// TwinCAT 3 PLC project TcUnit
// Title: TcUnit
// Company: www.tcunit.org
// Author: Jakob Sagatowski and contributors
// ProjectVersion: 1.0.1.1
// Description: TwinCAT unit testing framework. Documentation and examples are available at www.tcunit.org
// ProgramVersion: 3.1.4023.0
// libraries:
//   SysFile, * (System)
//   Tc2_Standard, * (Beckhoff Automation GmbH)
//   Tc2_System, * (Beckhoff Automation GmbH)
//   Tc2_Utilities, * (Beckhoff Automation GmbH)
//   Base Interfaces,newest,System
// project tree:
//   DUTs/ E_XmlError.TcDUT (not stored), ST_ADSLogStringMessage.TcDUT (not stored), ST_AssertResult.TcDUT (not stored), ST_AssertResultInstances.TcDUT (not stored), ST_AssertArrayResult.TcDUT (not stored), ST_AssertArrayResultInstances.TcDUT (not stored), U_ExpectedOrActual.TcDUT (not stored)
//   GVLs/ GVL_Param_TcUnit.TcGVL (not stored), GVL_Param_XmlControl.TcGVL (not stored), GVL_TcUnit.TcGVL (not stored)
//   ITFs/ I_AssertMessageFormatter.TcIO (not stored), I_TestResultFormatter.TcIO (not stored)
//   POUs/ FB_StringBuffer.TcPOU (not stored), FB_XmlControl.TcPOU (not stored), FB_FileControl.TcPOU (not stored), FB_AdjustAssertFailureMessageToMax252CharLength.TcPOU (not stored), FB_ADSAssertMessageFormatter.TcPOU (not stored), FB_ADSLogStringMessageFifoQueue.TcPOU (not stored), FB_ADSTestResultFormatter.TcPOU (not stored), FB_AnyComparator.TcPOU (not stored), FB_AssertResultStatic.TcPOU (not stored), FB_AssertArrayResultStatic.TcPOU (not stored), FB_TcUnitRunner.TcPOU (not stored), FB_Test.TcPOU (not stored), FB_TestSuite.TcPOU
//   POUs/Functions/ F_AnyToUnionValue.TcPOU (not stored), F_AnyTypeClassToString.TcPOU (not stored), F_IsAnyEqualToUnionValue.TcPOU (not stored), F_RemoveInstancePathAndProjectNameFromTestInstancePath.TcPOU (not stored), IS_TEST_FINISHED.TcPOU (not stored), RUN.TcPOU (not stored), TEST.TcPOU (not stored), TEST_FINISHED.TcPOU (not stored), TEST_FINISHED_NAMED.TcPOU (not stored)
//   POUs/Functions/WRITE_PROTECTED_/ WRITE_PROTECTED_BOOL.TcPOU (not stored), WRITE_PROTECTED_BYTE.TcPOU (not stored), WRITE_PROTECTED_DATE.TcPOU (not stored), WRITE_PROTECTED_DATE_AND_TIME.TcPOU (not stored), WRITE_PROTECTED_DINT.TcPOU (not stored), WRITE_PROTECTED_DWORD.TcPOU (not stored), WRITE_PROTECTED_INT.TcPOU (not stored), WRITE_PROTECTED_LREAL.TcPOU (not stored), WRITE_PROTECTED_REAL.TcPOU (not stored), WRITE_PROTECTED_SINT.TcPOU (not stored), WRITE_PROTECTED_STRING.TcPOU (not stored), WRITE_PROTECTED_TIME.TcPOU (not stored), WRITE_PROTECTED_TIME_OF_DAY.TcPOU (not stored), WRITE_PROTECTED_UDINT.TcPOU (not stored), WRITE_PROTECTED_UINT.TcPOU (not stored), WRITE_PROTECTED_USINT.TcPOU (not stored), WRITE_PROTECTED_WORD.TcPOU (not stored)
//   Version/ Global_Version.TcGVL

// ---- Version/Global_Version.TcGVL
{attribute 'TcGenerated'}
{attribute 'no-analysis'}
{attribute 'linkalways'}
// This function has been automatically generated from the project information.
VAR_GLOBAL CONSTANT
	{attribute 'const_non_replaced'}
	stLibVersion_TcUnit : ST_LibVersion := (iMajor := 1, iMinor := 0, iBuild := 1, iRevision := 1, nFlags := 0, sVersion := '1.0.1.1');
END_VAR

// ---- POUs/FB_TestSuite.TcPOU
(* This function block is responsible for holding the internal state of the test suite.
   Every test suite can have one or more tests, and every test can do one or more asserts.
   It's also responsible for providing all the assert-methods for asserting different data types.
   Only failed assertions are recorded.
*)
{attribute 'call_after_init'}
{attribute 'reflection'}
FUNCTION_BLOCK FB_TestSuite
VAR
    {attribute 'instance-path'}
    {attribute 'noinit'}
    InstancePath : Tc2_System.T_MaxString;

    (* We need to have access to specific information of the current task that this test suite
       is executed in. This is for instance necessary when we need to know whether a test is
       defined already. The definition of a test that is defined already is that we call on it
       with the same name twice in the same cycle *)
    GetCurrentTaskIndex : Tc2_System.GETCURTASKINDEX;

    NumberOfTests : UINT := 0;
    Tests : ARRAY[1..GVL_Param_TcUnit.MaxNumberOfTestsForEachTestSuite] OF FB_Test;
    (* Rising trigger of whether we have already notified the user of that the test name pointed to by the current
       position is a duplicate *)
    TestDuplicateNameTrigger : ARRAY[1..GVL_Param_TcUnit.MaxNumberOfTestsForEachTestSuite] OF Tc2_Standard.R_TRIG;
    (* Last cycle count index for a specific test. Used to detect whether this test has already been defined in the
       current test suite *)
    TestCycleCountIndex : ARRAY[1..GVL_Param_TcUnit.MaxNumberOfTestsForEachTestSuite] OF UDINT;

    AssertResults : FB_AssertResultStatic;
    AssertArrayResult : FB_AssertArrayResultStatic;

    (* Prints the failed asserts to ADS so that Visual Studio can display the assert message.
       This assert formatter can be replaced with something else than ADS *)
    ADSAssertMessageFormatter : FB_ADSAssertMessageFormatter;
    AssertMessageFormatter : I_AssertMessageFormatter := ADSAssertMessageFormatter;
END_VAR

METHOD PUBLIC AddTest
VAR_INPUT
    TestName : Tc2_System.T_MaxString;
END_VAR
VAR
    IteratorCounter : UINT;
    ErrorMessage : Tc2_System.T_MaxString;
    TestInstancePath : Tc2_System.T_MaxString;
    FunctionCallResult : DINT;
    CycleCount : UDINT;
    TestWithThisNameAlreadyExists : BOOL := FALSE;
    LowerCasedTestName : Tc2_System.T_MaxString;
    TrimmedTestName : Tc2_System.T_MaxString;
END_VAR
GVL_TcUnit.IgnoreCurrentTest := FALSE; // Reset the ignore current test flag

TrimmedTestName := Tc2_Utilities.F_LTrim(in := TestName);
TrimmedTestName := Tc2_Utilities.F_RTrim(in := TrimmedTestName);
LowerCasedTestName := Tc2_Utilities.F_ToLCase(in := TrimmedTestName);

(* Check if this test should be disabled *)
IF Tc2_Utilities.FIND(STR1 := LowerCasedTestName, STR2 := 'disabled_') = 1 THEN
    GVL_TcUnit.IgnoreCurrentTest := TRUE;
    RETURN;
END_IF

GetCurrentTaskIndex(); // Gets the task index of where this function block instance is being run in

(* Check if the test name already exists. Make sure there are no other tests with the same name already
   added for this test suite *)

CycleCount := TwinCAT_SystemInfoVarList._TaskInfo[GetCurrentTaskIndex.index].CycleCount;

(* Iterate all the test names that up to this point have been added for this test suite *)
FOR IteratorCounter := 1 TO NumberOfTests BY 1 DO
    IF Tests[IteratorCounter].GetName() = TrimmedTestName THEN
        TestWithThisNameAlreadyExists := TRUE;
        (* Check if a test with this name has already been called in this PLC cycle *)
        IF TestCycleCountIndex[IteratorCounter] = CycleCount THEN
            GVL_TcUnit.IgnoreCurrentTest := TRUE;
            (* A test with this name already exists for this test suite and has already been called in this cycle.
               Send a message notification, but only if we have not done so already. *)
            TestDuplicateNameTrigger[IteratorCounter](CLK := TRUE);
            IF TestDuplicateNameTrigger[IteratorCounter].Q THEN // Rising edge detected. We have not reported this before
                TestInstancePath := F_RemoveInstancePathAndProjectNameFromTestInstancePath(TestInstancePath :=
                                                                                           GVL_TcUnit.CurrentTestSuiteBeingCalled^.GetInstancePath());
                ErrorMessage := 'Test with name $'%s$' already exists in test suite $'';
                ErrorMessage := Tc2_Standard.CONCAT(STR1 := ErrorMessage, STR2 := TestInstancePath);
                ErrorMessage := Tc2_Standard.CONCAT(STR1 := ErrorMessage, STR2 := '$'');
                GVL_TcUnit.AdsLogger.WriteLog(MsgFmtStr := ErrorMessage,
                                              StrArg := TrimmedTestName);
            END_IF
        END_IF
        TestCycleCountIndex[IteratorCounter] := CycleCount;
    END_IF
END_FOR

IF NOT TestWithThisNameAlreadyExists THEN
    (* Test has not been found. Add it. *)
    Tests[IteratorCounter].SetName(Name := TrimmedTestName);
    NumberOfTests := NumberOfTests + 1;
    TestCycleCountIndex[NumberOfTests] := CycleCount;
END_IF
END_METHOD

METHOD PRIVATE AddTestNameToInstancePath : Tc2_System.T_MaxString
VAR_INPUT
    TestInstancePath : Tc2_System.T_MaxString;
END_VAR
VAR
    CompleteTestInstancePath : Tc2_System.T_MaxString;
END_VAR
CompleteTestInstancePath := Tc2_Utilities.CONCAT(STR1 := TestInstancePath, STR2 := '@');
AddTestNameToInstancePath := Tc2_Utilities.CONCAT(STR1 := CompleteTestInstancePath, STR2 := GVL_TcUnit.CurrentTestNameBeingCalled);
END_METHOD

METHOD PUBLIC AreAllTestsFinished : BOOL
VAR
    Counter : UINT;

    GetCurTaskIndex : Tc2_System.GETCURTASKINDEX;
END_VAR
AreAllTestsFinished := FALSE;

IF NumberOfTests > 0 THEN
    AreAllTestsFinished := TRUE;
    FOR Counter := 1 TO GetNumberOfTests() BY 1 DO
        AreAllTestsFinished := AreAllTestsFinished AND Tests[Counter].IsFinished();
    END_FOR
END_IF

(* If we have been running at least one cycle and no tests are registered it means that this testsuite is empty
   and doesn't contain any test cases. In that case, add a warning message and ignore this testsuite. *)
GetCurTaskIndex();
IF NumberOfTests = 0 AND NOT TwinCAT_SystemInfoVarList._TaskInfo[GetCurTaskIndex.index].FirstCycle THEN
    AreAllTestsFinished := TRUE;
END_IF
END_METHOD

METHOD PUBLIC AssertArray2dEquals_LREAL
VAR_IN_OUT
    Expecteds : ARRAY[*,*] OF LREAL; // LREAL 2d array with expected values
    Actuals : ARRAY[*,*] OF LREAL; // LREAL 2d array with actual values
END_VAR
VAR_INPUT
    Delta : LREAL; // The maximum delta between the value of expected and actual for which both numbers are still considered equal, proportional to the Expected value in that array cell
    Message : Tc2_System.T_MaxString; // The identifying message for the assertion error
END_VAR
VAR
    Equals : BOOL := TRUE;
    SizeEquals : BOOL := TRUE;
    ExpectedString : STRING;
    ActualString : STRING;
    AlreadyReported : BOOL;
    TestInstancePath : Tc2_System.T_MaxString;
    DimensionIndex : USINT; // Index when looping through Dimensions
    LowerBoundExpecteds : ARRAY[1..2] OF DINT; // Lower bounds of Expecteds array in each dimension
    UpperBoundExpecteds : ARRAY[1..2] OF DINT; // Upper bounds of Expecteds array in each dimension
    LowerBoundActuals : ARRAY[1..2] OF DINT; // Lower bounds of Actuals array in each dimension
    UpperBoundActuals : ARRAY[1..2] OF DINT; // Upper bounds of Actuals array in each dimension
    SizeOfExpecteds : ARRAY[1..2] OF DINT; // Size of Expecteds array in each dimension
    SizeOfActuals : ARRAY[1..2] OF DINT; // Size of Actuals array in each dimension
    Offset : ARRAY[1..2] OF DINT; // Current Array index offsets from Lower Bound in each dimension
    ExpectedArrayIndex : ARRAY[1..2] OF DINT; // Array of current Expected array indexes when looping through arrays
    ActualArrayIndex : ARRAY[1..2] OF DINT; // Array of current Actual array indexes when looping through arrays
    Expected : LREAL; // Single expected value
    Actual : LREAL; // Single actual value
END_VAR
IF GVL_TcUnit.IgnoreCurrentTest OR GVL_TcUnit.CurrentTestIsFinished THEN
    RETURN;
END_IF

TestInstancePath := AddTestNameToInstancePath(FindTestSuiteInstancePath());

(* UPPER_BOUND and LOWER_BOUND require literals for their second parameter,
   so they can't be called in a dimension-based loop.
   Thus we copy the array dimensions into arrays which accept variable indexes *)
LowerBoundExpecteds[1] := LOWER_BOUND(Expecteds, 1);
UpperBoundExpecteds[1] := UPPER_BOUND(Expecteds, 1);
LowerBoundExpecteds[2] := LOWER_BOUND(Expecteds, 2);
UpperBoundExpecteds[2] := UPPER_BOUND(Expecteds, 2);
LowerBoundActuals[1] := LOWER_BOUND(Actuals, 1);
UpperBoundActuals[1] := UPPER_BOUND(Actuals, 1);
LowerBoundActuals[2] := LOWER_BOUND(Actuals, 2);
UpperBoundActuals[2] := UPPER_BOUND(Actuals, 2);

FOR DimensionIndex := 1 TO 2 DO
    SizeOfExpecteds[DimensionIndex] := ABS(UpperBoundExpecteds[DimensionIndex] - LowerBoundExpecteds[DimensionIndex]) + 1;
    SizeOfActuals[DimensionIndex] := ABS(UpperBoundActuals[DimensionIndex] - LowerBoundActuals[DimensionIndex]) + 1;

    IF SizeOfExpecteds[DimensionIndex] <> SizeOfActuals[DimensionIndex] THEN
        Equals := FALSE;
        SizeEquals := FALSE;
    END_IF
END_FOR

IF SizeEquals THEN
    (* Even though we know that both arrays are equal in size, the two arrays can start at two completely different
       indexes in each dimension, which needs to be taken into account. *)
    FOR Offset[1] := 0 TO SizeOfExpecteds[1] - 1 DO // Iterate Dimension 1
        FOR Offset[2] := 0 TO SizeOfExpecteds[2] - 1 DO // Iterate Dimension 2
            // Update index variables
            FOR DimensionIndex := 1 TO 2 DO
                ExpectedArrayIndex[DimensionIndex] := LowerBoundExpecteds[DimensionIndex] + Offset[DimensionIndex];
                ActualArrayIndex[DimensionIndex] := LowerBoundActuals[DimensionIndex] + Offset[DimensionIndex];
            END_FOR

            // Get array element values
            Expected := Expecteds[ExpectedArrayIndex[1], ExpectedArrayIndex[2]];
            Actual := Actuals[ActualArrayIndex[1], ActualArrayIndex[2]]; 

            IF ABS(Expected - Actual) > Delta THEN
                Equals := FALSE;
                EXIT;
            END_IF
        END_FOR

        // Check for loop bailout
        IF NOT Equals THEN
            EXIT;
        END_IF
    END_FOR
END_IF

IF NOT Equals THEN
    AssertArrayResult.ReportResult(ExpectedsSize := DINT_TO_UDINT(SizeOfExpecteds[1] * SizeOfExpecteds[2]),
                                   ExpectedsTypeClass := IBaseLibrary.TypeClass.TYPE_LREAL,
                                   ActualsSize := DINT_TO_UDINT(SizeOfActuals[1] * SizeOfActuals[2]),
                                   ActualsTypeClass := IBaseLibrary.TypeClass.TYPE_LREAL,
                                   Message := Message,
                                   TestInstancePath := TestInstancePath,
                                   AlreadyReported => AlreadyReported);
END_IF

IF NOT AlreadyReported AND NOT Equals THEN
    SetTestFailed();

    IF NOT SizeEquals THEN
        Message := Tc2_Standard.CONCAT(STR1 := Message, STR2 := ', size of arrays not matching.');
        ExpectedString := 'SIZE = [';
        ExpectedString := Tc2_Standard.CONCAT(STR1 := ExpectedString, STR2 := DINT_TO_STRING(LowerBoundExpecteds[1]));
        ExpectedString := Tc2_Standard.CONCAT(STR1 := ExpectedString, STR2 := '..');
        ExpectedString := Tc2_Standard.CONCAT(STR1 := ExpectedString, STR2 := DINT_TO_STRING(UpperBoundExpecteds[1]));
        ExpectedString := Tc2_Standard.CONCAT(STR1 := ExpectedString, STR2 := ',');
        ExpectedString := Tc2_Standard.CONCAT(STR1 := ExpectedString, STR2 := DINT_TO_STRING(LowerBoundExpecteds[2]));
        ExpectedString := Tc2_Standard.CONCAT(STR1 := ExpectedString, STR2 := '..');
        ExpectedString := Tc2_Standard.CONCAT(STR1 := ExpectedString, STR2 := DINT_TO_STRING(UpperBoundExpecteds[2]));
        ExpectedString := Tc2_Standard.CONCAT(STR1 := ExpectedString, STR2 := '] (');
        ExpectedString := Tc2_Standard.CONCAT(STR1 := ExpectedString, STR2 := DINT_TO_STRING(SizeOfExpecteds[1]));
        ExpectedString := Tc2_Standard.CONCAT(STR1 := ExpectedString, STR2 := 'x');
        ExpectedString := Tc2_Standard.CONCAT(STR1 := ExpectedString, STR2 := DINT_TO_STRING(SizeOfExpecteds[2]));
        ExpectedString := Tc2_Standard.CONCAT(STR1 := ExpectedString, STR2 := ')');

        ActualString := 'SIZE = [';
        ActualString := Tc2_Standard.CONCAT(STR1 := ActualString, STR2 := DINT_TO_STRING(LowerBoundActuals[1]));
        ActualString := Tc2_Standard.CONCAT(STR1 := ActualString, STR2 := '..');
        ActualString := Tc2_Standard.CONCAT(STR1 := ActualString, STR2 := DINT_TO_STRING(UpperBoundActuals[1]));
        ActualString := Tc2_Standard.CONCAT(STR1 := ActualString, STR2 := ',');
        ActualString := Tc2_Standard.CONCAT(STR1 := ActualString, STR2 := DINT_TO_STRING(LowerBoundActuals[2]));
        ActualString := Tc2_Standard.CONCAT(STR1 := ActualString, STR2 := '..');
        ActualString := Tc2_Standard.CONCAT(STR1 := ActualString, STR2 := DINT_TO_STRING(UpperBoundActuals[2]));
        ActualString := Tc2_Standard.CONCAT(STR1 := ActualString, STR2 := '] (');
        ActualString := Tc2_Standard.CONCAT(STR1 := ActualString, STR2 := DINT_TO_STRING(SizeOfActuals[1]));
        ActualString := Tc2_Standard.CONCAT(STR1 := ActualString, STR2 := 'x');
        ActualString := Tc2_Standard.CONCAT(STR1 := ActualString, STR2 := DINT_TO_STRING(SizeOfActuals[2]));
        ActualString := Tc2_Standard.CONCAT(STR1 := ActualString, STR2 := ')');
    ELSE
        ExpectedString := 'ARRAY[';
        ExpectedString := Tc2_Standard.CONCAT(STR1 := ExpectedString, STR2 := DINT_TO_STRING(ExpectedArrayIndex[1]));
        ExpectedString := Tc2_Standard.CONCAT(STR1 := ExpectedString, STR2 := ',');
        ExpectedString := Tc2_Standard.CONCAT(STR1 := ExpectedString, STR2 := DINT_TO_STRING(ExpectedArrayIndex[2]));
        ExpectedString := Tc2_Standard.CONCAT(STR1 := ExpectedString, STR2 := '] = ');
        ExpectedString := Tc2_Standard.CONCAT(STR1 := ExpectedString, STR2 := LREAL_TO_STRING(Expected));

        ActualString := 'ARRAY[';
        ActualString := Tc2_Standard.CONCAT(STR1 := ActualString, STR2 := DINT_TO_STRING(ActualArrayIndex[1]));
        ActualString := Tc2_Standard.CONCAT(STR1 := ActualString, STR2 := ',');
        ActualString := Tc2_Standard.CONCAT(STR1 := ActualString, STR2 := DINT_TO_STRING(ActualArrayIndex[2]));
        ActualString := Tc2_Standard.CONCAT(STR1 := ActualString, STR2 := '] = ');
        ActualString := Tc2_Standard.CONCAT(STR1 := ActualString, STR2 := LREAL_TO_STRING(Actual));
    END_IF

    AssertMessageFormatter.LogAssertFailure(Expected := ExpectedString,
                                            Actual := ActualString,
                                            Message := Message,
                                            TestInstancePath := TestInstancePath);
END_IF
END_METHOD

METHOD PUBLIC AssertArray2dEquals_REAL
VAR_IN_OUT
    Expecteds : ARRAY[*,*] OF REAL; // REAL 2d array with expected values
    Actuals : ARRAY[*,*] OF REAL; // REAL 2d array with actual values
END_VAR
VAR_INPUT
    Delta : REAL; // The maximum delta between the value of expected and actual for which both numbers are still considered equal, proportional to the Expected value in that array cell
    Message : Tc2_System.T_MaxString; // The identifying message for the assertion error
END_VAR
VAR
    Equals : BOOL := TRUE;
    SizeEquals : BOOL := TRUE;
    ExpectedString : STRING;
    ActualString : STRING;
    AlreadyReported : BOOL;
    TestInstancePath : Tc2_System.T_MaxString;
    DimensionIndex : USINT; // Index when looping through Dimensions
    LowerBoundExpecteds : ARRAY[1..2] OF DINT; // Lower bounds of Expecteds array in each dimension
    UpperBoundExpecteds : ARRAY[1..2] OF DINT; // Upper bounds of Expecteds array in each dimension
    LowerBoundActuals : ARRAY[1..2] OF DINT; // Lower bounds of Actuals array in each dimension
    UpperBoundActuals : ARRAY[1..2] OF DINT; // Upper bounds of Actuals array in each dimension
    SizeOfExpecteds : ARRAY[1..2] OF DINT; // Size of Expecteds array in each dimension
    SizeOfActuals : ARRAY[1..2] OF DINT; // Size of Actuals array in each dimension
    Offset : ARRAY[1..2] OF DINT; // Current Array index offsets from Lower Bound in each dimension
    ExpectedArrayIndex : ARRAY[1..2] OF DINT; // Array of current Expected array indexes when looping through arrays
    ActualArrayIndex : ARRAY[1..2] OF DINT; // Array of current Actual array indexes when looping through arrays
    Expected : REAL; // Single expected value
    Actual : REAL; // Single actual value
END_VAR
IF GVL_TcUnit.IgnoreCurrentTest OR GVL_TcUnit.CurrentTestIsFinished THEN
    RETURN;
END_IF

TestInstancePath := AddTestNameToInstancePath(FindTestSuiteInstancePath());

(* UPPER_BOUND and LOWER_BOUND require literals for their second parameter, 
   so they can't be called in a dimension-based loop.
   Thus we copy the ARRAY dimensions into arrays which accept variable indexes *)
LowerBoundExpecteds[1] := LOWER_BOUND(Expecteds, 1);
UpperBoundExpecteds[1] := UPPER_BOUND(Expecteds, 1);
LowerBoundExpecteds[2] := LOWER_BOUND(Expecteds, 2);
UpperBoundExpecteds[2] := UPPER_BOUND(Expecteds, 2);
LowerBoundActuals[1] := LOWER_BOUND(Actuals, 1);
UpperBoundActuals[1] := UPPER_BOUND(Actuals, 1);
LowerBoundActuals[2] := LOWER_BOUND(Actuals, 2);
UpperBoundActuals[2] := UPPER_BOUND(Actuals, 2);

FOR DimensionIndex := 1 TO 2 DO
    SizeOfExpecteds[DimensionIndex] := ABS(UpperBoundExpecteds[DimensionIndex] - LowerBoundExpecteds[DimensionIndex]) + 1;
    SizeOfActuals[DimensionIndex] := ABS(UpperBoundActuals[DimensionIndex] - LowerBoundActuals[DimensionIndex]) + 1;

    IF SizeOfExpecteds[DimensionIndex] <> SizeOfActuals[DimensionIndex] THEN
        Equals := FALSE;
        SizeEquals := FALSE;
    END_IF
END_FOR

IF SizeEquals THEN
    (* Even though we know that both arrays are equal in size, the two arrays can start at two completely different
       indexes in each dimension, which needs to be taken into account. *)
    FOR Offset[1] := 0 TO SizeOfExpecteds[1] - 1 DO // Iterate Dimension 1
        FOR Offset[2] := 0 TO SizeOfExpecteds[2] - 1 DO // Iterate Dimension 2
            // Update index variables
            FOR DimensionIndex := 1 TO 2 DO
                ExpectedArrayIndex[DimensionIndex] := LowerBoundExpecteds[DimensionIndex] + Offset[DimensionIndex];
                ActualArrayIndex[DimensionIndex] := LowerBoundActuals[DimensionIndex] + Offset[DimensionIndex];
            END_FOR

            // Get array element values
            Expected := Expecteds[ExpectedArrayIndex[1], ExpectedArrayIndex[2]];
            Actual := Actuals[ActualArrayIndex[1], ActualArrayIndex[2]]; 

            IF ABS(Expected - Actual) > Delta THEN
                Equals := FALSE;
                EXIT;
            END_IF
        END_FOR

        // Check for loop bailout
        IF NOT Equals THEN
            EXIT;
        END_IF
    END_FOR
END_IF

IF NOT Equals THEN
    AssertArrayResult.ReportResult(ExpectedsSize := DINT_TO_UDINT(SizeOfExpecteds[1] * SizeOfExpecteds[2]),
                                   ExpectedsTypeClass := IBaseLibrary.TypeClass.TYPE_REAL,
                                   ActualsSize := DINT_TO_UDINT(SizeOfActuals[1] * SizeOfActuals[2]),
                                   ActualsTypeClass := IBaseLibrary.TypeClass.TYPE_REAL,
                                   Message := Message,
                                   TestInstancePath := TestInstancePath,
                                   AlreadyReported => AlreadyReported);
END_IF

IF NOT AlreadyReported AND NOT Equals THEN
    SetTestFailed();

    IF NOT SizeEquals THEN
        Message := Tc2_Standard.CONCAT(STR1 := Message, STR2 := ', size of arrays not matching.');
        ExpectedString := 'SIZE = [';
        ExpectedString := Tc2_Standard.CONCAT(STR1 := ExpectedString, STR2 := DINT_TO_STRING(LowerBoundExpecteds[1]));
        ExpectedString := Tc2_Standard.CONCAT(STR1 := ExpectedString, STR2 := '..');
        ExpectedString := Tc2_Standard.CONCAT(STR1 := ExpectedString, STR2 := DINT_TO_STRING(UpperBoundExpecteds[1]));
        ExpectedString := Tc2_Standard.CONCAT(STR1 := ExpectedString, STR2 := ',');
        ExpectedString := Tc2_Standard.CONCAT(STR1 := ExpectedString, STR2 := DINT_TO_STRING(LowerBoundExpecteds[2]));
        ExpectedString := Tc2_Standard.CONCAT(STR1 := ExpectedString, STR2 := '..');
        ExpectedString := Tc2_Standard.CONCAT(STR1 := ExpectedString, STR2 := DINT_TO_STRING(UpperBoundExpecteds[2]));
        ExpectedString := Tc2_Standard.CONCAT(STR1 := ExpectedString, STR2 := '] (');
        ExpectedString := Tc2_Standard.CONCAT(STR1 := ExpectedString, STR2 := DINT_TO_STRING(SizeOfExpecteds[1]));
        ExpectedString := Tc2_Standard.CONCAT(STR1 := ExpectedString, STR2 := 'x');
        ExpectedString := Tc2_Standard.CONCAT(STR1 := ExpectedString, STR2 := DINT_TO_STRING(SizeOfExpecteds[2]));
        ExpectedString := Tc2_Standard.CONCAT(STR1 := ExpectedString, STR2 := ')');

        ActualString := 'SIZE = [';
        ActualString := Tc2_Standard.CONCAT(STR1 := ActualString, STR2 := DINT_TO_STRING(LowerBoundActuals[1]));
        ActualString := Tc2_Standard.CONCAT(STR1 := ActualString, STR2 := '..');
        ActualString := Tc2_Standard.CONCAT(STR1 := ActualString, STR2 := DINT_TO_STRING(UpperBoundActuals[1]));
        ActualString := Tc2_Standard.CONCAT(STR1 := ActualString, STR2 := ',');
        ActualString := Tc2_Standard.CONCAT(STR1 := ActualString, STR2 := DINT_TO_STRING(LowerBoundActuals[2]));
        ActualString := Tc2_Standard.CONCAT(STR1 := ActualString, STR2 := '..');
        ActualString := Tc2_Standard.CONCAT(STR1 := ActualString, STR2 := DINT_TO_STRING(UpperBoundActuals[2]));
        ActualString := Tc2_Standard.CONCAT(STR1 := ActualString, STR2 := '] (');
        ActualString := Tc2_Standard.CONCAT(STR1 := ActualString, STR2 := DINT_TO_STRING(SizeOfActuals[1]));
        ActualString := Tc2_Standard.CONCAT(STR1 := ActualString, STR2 := 'x');
        ActualString := Tc2_Standard.CONCAT(STR1 := ActualString, STR2 := DINT_TO_STRING(SizeOfActuals[2]));
        ActualString := Tc2_Standard.CONCAT(STR1 := ActualString, STR2 := ')');
    ELSE
        ExpectedString := 'ARRAY[';
        ExpectedString := Tc2_Standard.CONCAT(STR1 := ExpectedString, STR2 := DINT_TO_STRING(ExpectedArrayIndex[1]));
        ExpectedString := Tc2_Standard.CONCAT(STR1 := ExpectedString, STR2 := ',');
        ExpectedString := Tc2_Standard.CONCAT(STR1 := ExpectedString, STR2 := DINT_TO_STRING(ExpectedArrayIndex[2]));
        ExpectedString := Tc2_Standard.CONCAT(STR1 := ExpectedString, STR2 := '] = ');
        ExpectedString := Tc2_Standard.CONCAT(STR1 := ExpectedString, STR2 := REAL_TO_STRING(Expected));

        ActualString := 'ARRAY[';
        ActualString := Tc2_Standard.CONCAT(STR1 := ActualString, STR2 := DINT_TO_STRING(ActualArrayIndex[1]));
        ActualString := Tc2_Standard.CONCAT(STR1 := ActualString, STR2 := ',');
        ActualString := Tc2_Standard.CONCAT(STR1 := ActualString, STR2 := DINT_TO_STRING(ActualArrayIndex[2]));
        ActualString := Tc2_Standard.CONCAT(STR1 := ActualString, STR2 := '] = ');
        ActualString := Tc2_Standard.CONCAT(STR1 := ActualString, STR2 := REAL_TO_STRING(Actual));
    END_IF

    AssertMessageFormatter.LogAssertFailure(Expected := ExpectedString,
                                            Actual := ActualString,
                                            Message := Message,
                                            TestInstancePath := TestInstancePath);
END_IF
END_METHOD

METHOD PUBLIC AssertArray3dEquals_LREAL
VAR_IN_OUT
    Expecteds : ARRAY[*,*,*] OF LREAL; // LREAL 3d array with expected values
    Actuals : ARRAY[*,*,*] OF LREAL; // LREAL 3d array with actual values
END_VAR
VAR_INPUT
    Delta : LREAL;  // The maximum delta between the value of expected and actual for which both numbers are still considered equal, proportional to the Expected value in that array cell
    Message : Tc2_System.T_MaxString; // The identifying message for the assertion error
END_VAR
VAR
    Equals : BOOL := TRUE;
    SizeEquals : BOOL := TRUE;
    ExpectedString : STRING;
    ActualString : STRING;
    AlreadyReported : BOOL;
    TestInstancePath : Tc2_System.T_MaxString;
    DimensionIndex : USINT;  // Index when looping through Dimensions
    LowerBoundExpecteds : ARRAY[1..3] OF DINT; // Lower bounds of Expecteds array in each dimension
    UpperBoundExpecteds : ARRAY[1..3] OF DINT; // Upper bounds of Expecteds array in each dimension
    LowerBoundActuals : ARRAY[1..3] OF DINT; // Lower bounds of Actuals array in each dimension
    UpperBoundActuals : ARRAY[1..3] OF DINT; // Upper bounds of Actuals array in each dimension
    SizeOfExpecteds : ARRAY[1..3] OF DINT; // Size of Expecteds array in each dimension
    SizeOfActuals : ARRAY[1..3] OF DINT; // Size of Actuals array in each dimension
    Offset : ARRAY[1..3] OF DINT; // Current Array index offsets from Lower Bound in each dimension
    ExpectedArrayIndex : ARRAY[1..3] OF DINT; // Array of current Expected array indexes when looping through arrays
    ActualArrayIndex : ARRAY[1..3] OF DINT; // Array of current Actual array indexes when looping through arrays
    Expected : LREAL; // Single expected value
    Actual : LREAL; // Single actual value
END_VAR
IF GVL_TcUnit.IgnoreCurrentTest OR GVL_TcUnit.CurrentTestIsFinished THEN
    RETURN;
END_IF

TestInstancePath := AddTestNameToInstancePath(FindTestSuiteInstancePath());

(* UPPER_BOUND and LOWER_BOUND require literals for their second parameter,
   so they can't be called in a dimension-based loop.
   Thus we copy the array dimensions into arrays which accept variable indexes *)
LowerBoundExpecteds[1] := LOWER_BOUND(Expecteds, 1);
UpperBoundExpecteds[1] := UPPER_BOUND(Expecteds, 1);
LowerBoundExpecteds[2] := LOWER_BOUND(Expecteds, 2);
UpperBoundExpecteds[2] := UPPER_BOUND(Expecteds, 2);
LowerBoundExpecteds[3] := LOWER_BOUND(Expecteds, 3);
UpperBoundExpecteds[3] := UPPER_BOUND(Expecteds, 3);
LowerBoundActuals[1] := LOWER_BOUND(Actuals, 1);
UpperBoundActuals[1] := UPPER_BOUND(Actuals, 1);
LowerBoundActuals[2] := LOWER_BOUND(Actuals, 2);
UpperBoundActuals[2] := UPPER_BOUND(Actuals, 2);
LowerBoundActuals[3] := LOWER_BOUND(Actuals, 3);
UpperBoundActuals[3] := UPPER_BOUND(Actuals, 3);

FOR DimensionIndex := 1 TO 3 DO
    SizeOfExpecteds[DimensionIndex] := ABS(UpperBoundExpecteds[DimensionIndex] - LowerBoundExpecteds[DimensionIndex]) + 1;
    SizeOfActuals[DimensionIndex] := ABS(UpperBoundActuals[DimensionIndex] - LowerBoundActuals[DimensionIndex]) + 1;

    IF SizeOfExpecteds[DimensionIndex] <> SizeOfActuals[DimensionIndex] THEN
        Equals := FALSE;
        SizeEquals := FALSE;
    END_IF
END_FOR

IF SizeEquals THEN
    (* Even though we know that both arrays are equal in size, the three arrays can start at three completely different
       indexes in each dimension, which needs to be taken into account. *)
    FOR Offset[1] := 0 TO SizeOfExpecteds[1] - 1 DO // Iterate Dimension 1
        FOR Offset[2] := 0 TO SizeOfExpecteds[2] - 1 DO // Iterate Dimension 2
            FOR Offset[3] := 0 TO SizeOfExpecteds[3] - 1 DO // Iterate Dimension 3
                // Update index variables
                FOR DimensionIndex := 1 TO 3 DO
                    ExpectedArrayIndex[DimensionIndex] := LowerBoundExpecteds[DimensionIndex] + Offset[DimensionIndex];
                    ActualArrayIndex[DimensionIndex] := LowerBoundActuals[DimensionIndex] + Offset[DimensionIndex];
                END_FOR

                // Get array element values
                Expected := Expecteds[ExpectedArrayIndex[1], ExpectedArrayIndex[2], ExpectedArrayIndex[3]];
                Actual := Actuals[ActualArrayIndex[1], ActualArrayIndex[2], ActualArrayIndex[3]]; 

                IF ABS(Expected - Actual) > Delta THEN
                    Equals := FALSE;
                    EXIT;
                END_IF
            END_FOR

            // Check for loop bailout
            IF NOT Equals THEN
                EXIT;
            END_IF
        END_FOR

        // Check for loop bailout
        IF NOT Equals THEN
            EXIT;
        END_IF
    END_FOR
END_IF

IF NOT Equals THEN
    AssertArrayResult.ReportResult(ExpectedsSize := DINT_TO_UDINT(SizeOfExpecteds[1] * SizeOfExpecteds[2] * SizeOfExpecteds[3]),
                                   ExpectedsTypeClass := IBaseLibrary.TypeClass.TYPE_LREAL,
                                   ActualsSize := DINT_TO_UDINT(SizeOfActuals[1] * SizeOfActuals[2] * SizeOfActuals[3]),
                                   ActualsTypeClass := IBaseLibrary.TypeClass.TYPE_LREAL,
                                   Message := Message,
                                   TestInstancePath := TestInstancePath,
                                   AlreadyReported => AlreadyReported);
END_IF

IF NOT AlreadyReported AND NOT Equals THEN
    SetTestFailed();

    IF NOT SizeEquals THEN
        Message := Tc2_Standard.CONCAT(STR1 := Message, STR2 := ', size of arrays not matching.');
        ExpectedString := 'SIZE = [';
        ExpectedString := Tc2_Standard.CONCAT(STR1 := ExpectedString, STR2 := DINT_TO_STRING(LowerBoundExpecteds[1]));
        ExpectedString := Tc2_Standard.CONCAT(STR1 := ExpectedString, STR2 := '..');
        ExpectedString := Tc2_Standard.CONCAT(STR1 := ExpectedString, STR2 := DINT_TO_STRING(UpperBoundExpecteds[1]));
        ExpectedString := Tc2_Standard.CONCAT(STR1 := ExpectedString, STR2 := ',');
        ExpectedString := Tc2_Standard.CONCAT(STR1 := ExpectedString, STR2 := DINT_TO_STRING(LowerBoundExpecteds[2]));
        ExpectedString := Tc2_Standard.CONCAT(STR1 := ExpectedString, STR2 := '..');
        ExpectedString := Tc2_Standard.CONCAT(STR1 := ExpectedString, STR2 := DINT_TO_STRING(UpperBoundExpecteds[2]));
        ExpectedString := Tc2_Standard.CONCAT(STR1 := ExpectedString, STR2 := ',');
        ExpectedString := Tc2_Standard.CONCAT(STR1 := ExpectedString, STR2 := DINT_TO_STRING(LowerBoundExpecteds[3]));
        ExpectedString := Tc2_Standard.CONCAT(STR1 := ExpectedString, STR2 := '..');
        ExpectedString := Tc2_Standard.CONCAT(STR1 := ExpectedString, STR2 := DINT_TO_STRING(UpperBoundExpecteds[3]));
        ExpectedString := Tc2_Standard.CONCAT(STR1 := ExpectedString, STR2 := '] (');
        ExpectedString := Tc2_Standard.CONCAT(STR1 := ExpectedString, STR2 := DINT_TO_STRING(SizeOfExpecteds[1]));
        ExpectedString := Tc2_Standard.CONCAT(STR1 := ExpectedString, STR2 := 'x');
        ExpectedString := Tc2_Standard.CONCAT(STR1 := ExpectedString, STR2 := DINT_TO_STRING(SizeOfExpecteds[2]));
        ExpectedString := Tc2_Standard.CONCAT(STR1 := ExpectedString, STR2 := 'x');
        ExpectedString := Tc2_Standard.CONCAT(STR1 := ExpectedString, STR2 := DINT_TO_STRING(SizeOfExpecteds[3]));
        ExpectedString := Tc2_Standard.CONCAT(STR1 := ExpectedString, STR2 := ')');

        ActualString := 'SIZE = [';
        ActualString := Tc2_Standard.CONCAT(STR1 := ActualString, STR2 := DINT_TO_STRING(LowerBoundActuals[1]));
        ActualString := Tc2_Standard.CONCAT(STR1 := ActualString, STR2 := '..');
        ActualString := Tc2_Standard.CONCAT(STR1 := ActualString, STR2 := DINT_TO_STRING(UpperBoundActuals[1]));
        ActualString := Tc2_Standard.CONCAT(STR1 := ActualString, STR2 := ',');
        ActualString := Tc2_Standard.CONCAT(STR1 := ActualString, STR2 := DINT_TO_STRING(LowerBoundActuals[2]));
        ActualString := Tc2_Standard.CONCAT(STR1 := ActualString, STR2 := '..');
        ActualString := Tc2_Standard.CONCAT(STR1 := ActualString, STR2 := DINT_TO_STRING(UpperBoundActuals[2]));
        ActualString := Tc2_Standard.CONCAT(STR1 := ActualString, STR2 := ',');
        ActualString := Tc2_Standard.CONCAT(STR1 := ActualString, STR2 := DINT_TO_STRING(LowerBoundActuals[3]));
        ActualString := Tc2_Standard.CONCAT(STR1 := ActualString, STR2 := '..');
        ActualString := Tc2_Standard.CONCAT(STR1 := ActualString, STR2 := DINT_TO_STRING(UpperBoundActuals[3]));
        ActualString := Tc2_Standard.CONCAT(STR1 := ActualString, STR2 := '] (');
        ActualString := Tc2_Standard.CONCAT(STR1 := ActualString, STR2 := DINT_TO_STRING(SizeOfActuals[1]));
        ActualString := Tc2_Standard.CONCAT(STR1 := ActualString, STR2 := 'x');
        ActualString := Tc2_Standard.CONCAT(STR1 := ActualString, STR2 := DINT_TO_STRING(SizeOfActuals[2]));
        ActualString := Tc2_Standard.CONCAT(STR1 := ActualString, STR2 := 'x');
        ActualString := Tc2_Standard.CONCAT(STR1 := ActualString, STR2 := DINT_TO_STRING(SizeOfActuals[3]));
        ActualString := Tc2_Standard.CONCAT(STR1 := ActualString, STR2 := ')');
    ELSE
        ExpectedString := 'ARRAY[';
        ExpectedString := Tc2_Standard.CONCAT(STR1 := ExpectedString, STR2 := DINT_TO_STRING(ExpectedArrayIndex[1]));
        ExpectedString := Tc2_Standard.CONCAT(STR1 := ExpectedString, STR2 := ',');
        ExpectedString := Tc2_Standard.CONCAT(STR1 := ExpectedString, STR2 := DINT_TO_STRING(ExpectedArrayIndex[2]));
        ExpectedString := Tc2_Standard.CONCAT(STR1 := ExpectedString, STR2 := ',');
        ExpectedString := Tc2_Standard.CONCAT(STR1 := ExpectedString, STR2 := DINT_TO_STRING(ExpectedArrayIndex[3]));
        ExpectedString := Tc2_Standard.CONCAT(STR1 := ExpectedString, STR2 := '] = ');
        ExpectedString := Tc2_Standard.CONCAT(STR1 := ExpectedString, STR2 := LREAL_TO_STRING(Expected) );

        ActualString := 'ARRAY[';
        ActualString := Tc2_Standard.CONCAT(STR1 := ActualString, STR2 := DINT_TO_STRING(ActualArrayIndex[1]));
        ActualString := Tc2_Standard.CONCAT(STR1 := ActualString, STR2 := ',');
        ActualString := Tc2_Standard.CONCAT(STR1 := ActualString, STR2 := DINT_TO_STRING(ActualArrayIndex[2]));
        ActualString := Tc2_Standard.CONCAT(STR1 := ActualString, STR2 := ',');
        ActualString := Tc2_Standard.CONCAT(STR1 := ActualString, STR2 := DINT_TO_STRING(ActualArrayIndex[3]));
        ActualString := Tc2_Standard.CONCAT(STR1 := ActualString, STR2 := '] = ');
        ActualString := Tc2_Standard.CONCAT(STR1 := ActualString, STR2 := LREAL_TO_STRING(Actual));
    END_IF

    AssertMessageFormatter.LogAssertFailure(Expected := ExpectedString,
                                            Actual := ActualString,
                                            Message := Message,
                                            TestInstancePath := TestInstancePath);
END_IF
END_METHOD

METHOD PUBLIC AssertArray3dEquals_REAL
VAR_IN_OUT
    Expecteds : ARRAY[*,*,*] OF REAL; // REAL 3d array with expected values
    Actuals : ARRAY[*,*,*] OF REAL; // REAL 3d array with actual values
END_VAR
VAR_INPUT
    Delta : REAL; // The maximum delta between the value of expected and actual for which both numbers are still considered equal, proportional to the Expected value in that array cell
    Message : Tc2_System.T_MaxString; // The identifying message for the assertion error
END_VAR
VAR
    Equals : BOOL := TRUE;
    SizeEquals : BOOL := TRUE;
    ExpectedString : STRING;
    ActualString : STRING;
    AlreadyReported : BOOL;
    TestInstancePath : Tc2_System.T_MaxString;
    DimensionIndex : USINT;  // Index when looping through Dimensions
    LowerBoundExpecteds : ARRAY[1..3] OF DINT; // Lower bounds of Expecteds array in each dimension
    UpperBoundExpecteds : ARRAY[1..3] OF DINT; // Upper bounds of Expecteds array in each dimension
    LowerBoundActuals : ARRAY[1..3] OF DINT; // Lower bounds of Actuals array in each dimension
    UpperBoundActuals : ARRAY[1..3] OF DINT; // Upper bounds of Actuals array in each dimension
    SizeOfExpecteds : ARRAY[1..3] OF DINT; // Size of Expecteds array in each dimension
    SizeOfActuals : ARRAY[1..3] OF DINT; // Size of Actuals array in each dimension
    Offset : ARRAY[1..3] OF DINT; // Current Array index offsets from Lower Bound in each dimension
    ExpectedArrayIndex : ARRAY[1..3] OF DINT; // Array of current Expected array indexes when looping through arrays
    ActualArrayIndex : ARRAY[1..3] OF DINT; // Array of current Actual array indexes when looping through arrays
    Expected : REAL; // Single expected value
    Actual : REAL; // Single actual value
    ExpectedValueString : Tc2_System.T_MaxString;
    ActualValueString : Tc2_System.T_MaxString;
    FormatString : Tc2_Utilities.FB_FormatString; // String formatter for output messages
END_VAR
IF GVL_TcUnit.IgnoreCurrentTest OR GVL_TcUnit.CurrentTestIsFinished THEN
    RETURN;
END_IF

TestInstancePath := AddTestNameToInstancePath(FindTestSuiteInstancePath());

(* UPPER_BOUND and LOWER_BOUND require literals for their second parameter,
   so they can't be called in a dimension-based loop.
   Thus we copy the array dimensions into arrays which accept variable indexes *)
LowerBoundExpecteds[1] := LOWER_BOUND(Expecteds, 1);
UpperBoundExpecteds[1] := UPPER_BOUND(Expecteds, 1);
LowerBoundExpecteds[2] := LOWER_BOUND(Expecteds, 2);
UpperBoundExpecteds[2] := UPPER_BOUND(Expecteds, 2);
LowerBoundExpecteds[3] := LOWER_BOUND(Expecteds, 3);
UpperBoundExpecteds[3] := UPPER_BOUND(Expecteds, 3);
LowerBoundActuals[1] := LOWER_BOUND(Actuals, 1);
UpperBoundActuals[1] := UPPER_BOUND(Actuals, 1);
LowerBoundActuals[2] := LOWER_BOUND(Actuals, 2);
UpperBoundActuals[2] := UPPER_BOUND(Actuals, 2);
LowerBoundActuals[3] := LOWER_BOUND(Actuals, 3);
UpperBoundActuals[3] := UPPER_BOUND(Actuals, 3);

FOR DimensionIndex := 1 TO 3 DO
    SizeOfExpecteds[DimensionIndex] := ABS(UpperBoundExpecteds[DimensionIndex] - LowerBoundExpecteds[DimensionIndex]) + 1;
    SizeOfActuals[DimensionIndex] := ABS(UpperBoundActuals[DimensionIndex] - LowerBoundActuals[DimensionIndex]) + 1;

    IF SizeOfExpecteds[DimensionIndex] <> SizeOfActuals[DimensionIndex] THEN
        Equals := FALSE;
        SizeEquals := FALSE;
    END_IF
END_FOR

IF SizeEquals THEN
    (* Even though we know that both arrays are equal in size, the two arrays can start at two completely different
       indexes in each dimension, which needs to be taken into account. *)
    FOR Offset[1] := 0 TO SizeOfExpecteds[1] - 1 DO // Iterate Dimension 1
        FOR Offset[2] := 0 TO SizeOfExpecteds[2] - 1 DO // Iterate Dimension 2
            FOR Offset[3] := 0 TO SizeOfExpecteds[3] - 1 DO // Iterate Dimension 3
                // Update index variables
                FOR DimensionIndex := 1 TO 3 DO
                    ExpectedArrayIndex[DimensionIndex] := LowerBoundExpecteds[DimensionIndex] + Offset[DimensionIndex];
                    ActualArrayIndex[DimensionIndex] := LowerBoundActuals[DimensionIndex] + Offset[DimensionIndex];
                END_FOR

                // Get array element values
                Expected := Expecteds[ExpectedArrayIndex[1], ExpectedArrayIndex[2], ExpectedArrayIndex[3]];
                Actual := Actuals[ActualArrayIndex[1], ActualArrayIndex[2], ActualArrayIndex[3]]; 

                IF ABS(Expected - Actual) > Delta THEN
                    Equals := FALSE;
                    EXIT;
                END_IF
            END_FOR

            // Check for loop bailout
            IF NOT Equals THEN
                EXIT;
            END_IF
        END_FOR

        // Check for loop bailout
        IF NOT Equals THEN
            EXIT;
        END_IF
    END_FOR
END_IF

IF NOT Equals THEN
    AssertArrayResult.ReportResult(ExpectedsSize := DINT_TO_UDINT(SizeOfExpecteds[1] * SizeOfExpecteds[2] * SizeOfExpecteds[3]),
                                   ExpectedsTypeClass := IBaseLibrary.TypeClass.TYPE_REAL,
                                   ActualsSize := DINT_TO_UDINT(SizeOfActuals[1] * SizeOfActuals[2] * SizeOfActuals[3]),
                                   ActualsTypeClass := IBaseLibrary.TypeClass.TYPE_REAL,
                                   Message := Message,
                                   TestInstancePath := TestInstancePath,
                                   AlreadyReported => AlreadyReported);
END_IF

IF NOT AlreadyReported AND NOT Equals THEN
    SetTestFailed();

    IF NOT SizeEquals THEN
        Message := Tc2_Standard.CONCAT(STR1 := Message, STR2 := ', size of arrays not matching.');
        ExpectedString := 'SIZE = [';
        ExpectedString := Tc2_Standard.CONCAT(STR1 := ExpectedString, STR2 := DINT_TO_STRING(LowerBoundExpecteds[1]));
        ExpectedString := Tc2_Standard.CONCAT(STR1 := ExpectedString, STR2 := '..');
        ExpectedString := Tc2_Standard.CONCAT(STR1 := ExpectedString, STR2 := DINT_TO_STRING(UpperBoundExpecteds[1]));
        ExpectedString := Tc2_Standard.CONCAT(STR1 := ExpectedString, STR2 := ',');
        ExpectedString := Tc2_Standard.CONCAT(STR1 := ExpectedString, STR2 := DINT_TO_STRING(LowerBoundExpecteds[2]));
        ExpectedString := Tc2_Standard.CONCAT(STR1 := ExpectedString, STR2 := '..');
        ExpectedString := Tc2_Standard.CONCAT(STR1 := ExpectedString, STR2 := DINT_TO_STRING(UpperBoundExpecteds[2]));
        ExpectedString := Tc2_Standard.CONCAT(STR1 := ExpectedString, STR2 := ',');
        ExpectedString := Tc2_Standard.CONCAT(STR1 := ExpectedString, STR2 := DINT_TO_STRING(LowerBoundExpecteds[3]));
        ExpectedString := Tc2_Standard.CONCAT(STR1 := ExpectedString, STR2 := '..');
        ExpectedString := Tc2_Standard.CONCAT(STR1 := ExpectedString, STR2 := DINT_TO_STRING(UpperBoundExpecteds[3]));
        ExpectedString := Tc2_Standard.CONCAT(STR1 := ExpectedString, STR2 := '] (');
        ExpectedString := Tc2_Standard.CONCAT(STR1 := ExpectedString, STR2 := DINT_TO_STRING(SizeOfExpecteds[1]));
        ExpectedString := Tc2_Standard.CONCAT(STR1 := ExpectedString, STR2 := 'x');
        ExpectedString := Tc2_Standard.CONCAT(STR1 := ExpectedString, STR2 := DINT_TO_STRING(SizeOfExpecteds[2]));
        ExpectedString := Tc2_Standard.CONCAT(STR1 := ExpectedString, STR2 := 'x');
        ExpectedString := Tc2_Standard.CONCAT(STR1 := ExpectedString, STR2 := DINT_TO_STRING(SizeOfExpecteds[3]));
        ExpectedString := Tc2_Standard.CONCAT(STR1 := ExpectedString, STR2 := ')');

        ActualString := 'SIZE = [';
        ActualString := Tc2_Standard.CONCAT(STR1 := ActualString, STR2 := DINT_TO_STRING(LowerBoundActuals[1]));
        ActualString := Tc2_Standard.CONCAT(STR1 := ActualString, STR2 := '..');
        ActualString := Tc2_Standard.CONCAT(STR1 := ActualString, STR2 := DINT_TO_STRING(UpperBoundActuals[1]));
        ActualString := Tc2_Standard.CONCAT(STR1 := ActualString, STR2 := ',');
        ActualString := Tc2_Standard.CONCAT(STR1 := ActualString, STR2 := DINT_TO_STRING(LowerBoundActuals[2]));
        ActualString := Tc2_Standard.CONCAT(STR1 := ActualString, STR2 := '..');
        ActualString := Tc2_Standard.CONCAT(STR1 := ActualString, STR2 := DINT_TO_STRING(UpperBoundActuals[2]));
        ActualString := Tc2_Standard.CONCAT(STR1 := ActualString, STR2 := ',');
        ActualString := Tc2_Standard.CONCAT(STR1 := ActualString, STR2 := DINT_TO_STRING(LowerBoundActuals[3]));
        ActualString := Tc2_Standard.CONCAT(STR1 := ActualString, STR2 := '..');
        ActualString := Tc2_Standard.CONCAT(STR1 := ActualString, STR2 := DINT_TO_STRING(UpperBoundActuals[3]));
        ActualString := Tc2_Standard.CONCAT(STR1 := ActualString, STR2 := '] (');
        ActualString := Tc2_Standard.CONCAT(STR1 := ActualString, STR2 := DINT_TO_STRING(SizeOfActuals[1]));
        ActualString := Tc2_Standard.CONCAT(STR1 := ActualString, STR2 := 'x');
        ActualString := Tc2_Standard.CONCAT(STR1 := ActualString, STR2 := DINT_TO_STRING(SizeOfActuals[2]));
        ActualString := Tc2_Standard.CONCAT(STR1 := ActualString, STR2 := 'x');
        ActualString := Tc2_Standard.CONCAT(STR1 := ActualString, STR2 := DINT_TO_STRING(SizeOfActuals[3]));
        ActualString := Tc2_Standard.CONCAT(STR1 := ActualString, STR2 := ')');
    ELSE
        ExpectedString := 'ARRAY[';
        ExpectedString := Tc2_Standard.CONCAT(STR1 := ExpectedString, STR2 := DINT_TO_STRING(ExpectedArrayIndex[1]));
        ExpectedString := Tc2_Standard.CONCAT(STR1 := ExpectedString, STR2 := ',');
        ExpectedString := Tc2_Standard.CONCAT(STR1 := ExpectedString, STR2 := DINT_TO_STRING(ExpectedArrayIndex[2]));
        ExpectedString := Tc2_Standard.CONCAT(STR1 := ExpectedString, STR2 := ',');
        ExpectedString := Tc2_Standard.CONCAT(STR1 := ExpectedString, STR2 := DINT_TO_STRING(ExpectedArrayIndex[3]));
        ExpectedString := Tc2_Standard.CONCAT(STR1 := ExpectedString, STR2 := '] = ');
        ExpectedString := Tc2_Standard.CONCAT(STR1 := ExpectedString, STR2 := REAL_TO_STRING(Expected) );

        ActualString := 'ARRAY[';
        ActualString := Tc2_Standard.CONCAT(STR1 := ActualString, STR2 := DINT_TO_STRING(ActualArrayIndex[1]));
        ActualString := Tc2_Standard.CONCAT(STR1 := ActualString, STR2 := ',');
        ActualString := Tc2_Standard.CONCAT(STR1 := ActualString, STR2 := DINT_TO_STRING(ActualArrayIndex[2]));
        ActualString := Tc2_Standard.CONCAT(STR1 := ActualString, STR2 := ',');
        ActualString := Tc2_Standard.CONCAT(STR1 := ActualString, STR2 := DINT_TO_STRING(ActualArrayIndex[3]));
        ActualString := Tc2_Standard.CONCAT(STR1 := ActualString, STR2 := '] = ');
        ActualString := Tc2_Standard.CONCAT(STR1 := ActualString, STR2 := REAL_TO_STRING(Actual));
    END_IF

    AssertMessageFormatter.LogAssertFailure(Expected := ExpectedString,
                                            Actual := ActualString,
                                            Message := Message,
                                            TestInstancePath := TestInstancePath);
END_IF
END_METHOD

(*
    Asserts that two BOOL arrays are equal. If they are not, an assertion error is created.
*)
METHOD PUBLIC AssertArrayEquals_BOOL
VAR_IN_OUT
    Expecteds : ARRAY[*] OF BOOL; // BOOL array with expected values
    Actuals : ARRAY[*] OF BOOL; // BOOL array with actual values
END_VAR
VAR_INPUT
    Message : Tc2_System.T_MaxString; // The identifying message for the assertion error
END_VAR
VAR
    Equals : BOOL := TRUE;
    SizeEquals : BOOL := TRUE;
    Index : DINT;
    ExpectedString : STRING;
    ActualString : STRING;
    AlreadyReported : BOOL;
    TestInstancePath : Tc2_System.T_MaxString;
    SizeOfExpecteds : DINT;
    SizeOfActuals : DINT;
    ExpectedsIndex : DINT;
    ActualsIndex : DINT;
END_VAR
IF GVL_TcUnit.IgnoreCurrentTest OR GVL_TcUnit.CurrentTestIsFinished THEN
    RETURN;
END_IF

TestInstancePath := AddTestNameToInstancePath(FindTestSuiteInstancePath());

SizeOfExpecteds := ABS(UPPER_BOUND(Expecteds, 1) - LOWER_BOUND(Expecteds, 1)) + 1;
SizeOfActuals := ABS(UPPER_BOUND(Actuals, 1) - LOWER_BOUND(Actuals, 1)) + 1;

IF SizeOfExpecteds <> SizeOfActuals THEN
    Equals := FALSE;
    SizeEquals := FALSE;
ELSE
    (* Even though we know that both arrays are equal in size, the two arrays can start at two completely different
       indexes, which needs to be taken into account for. *)
    ExpectedsIndex := LOWER_BOUND(Expecteds, 1); // The start position for the expecteds
    ActualsIndex := LOWER_BOUND(Actuals, 1); // The start position for the actuals
    FOR Index := 1 TO SizeOfExpecteds BY 1 DO
        IF Expecteds[ExpectedsIndex] <> Actuals[ActualsIndex] THEN
            Equals := FALSE;
            EXIT;
        END_IF
        ExpectedsIndex := ExpectedsIndex + 1;
        ActualsIndex := ActualsIndex + 1;
    END_FOR
END_IF

IF NOT Equals THEN
    AssertArrayResult.ReportResult(ExpectedsSize := DINT_TO_UDINT(SizeOfExpecteds),
                                   ExpectedsTypeClass := IBaseLibrary.TypeClass.TYPE_BOOL,
                                   ActualsSize := DINT_TO_UDINT(SizeOfActuals),
                                   ActualsTypeClass := IBaseLibrary.TypeClass.TYPE_BOOL,
                                   Message := Message,
                                   TestInstancePath := TestInstancePath,
                                   AlreadyReported => AlreadyReported);
END_IF

IF NOT AlreadyReported AND NOT Equals THEN
    SetTestFailed();
    
    IF NOT SizeEquals THEN
        Message := CONCAT(STR1 := Message, STR2 := ', size of arrays not matching.');
        ExpectedString := 'SIZE = ';
        ExpectedString := CONCAT(STR1 := ExpectedString, STR2 := DINT_TO_STRING(SizeOfExpecteds));
        ActualString := 'SIZE = ';
        ActualString := CONCAT(STR1 := ActualString, STR2 := DINT_TO_STRING(SizeOfActuals));
    ELSE
        ExpectedString := 'ARRAY[';
        ExpectedString := CONCAT(STR1 := ExpectedString, STR2 := DINT_TO_STRING(ExpectedsIndex));
        ExpectedString := CONCAT(STR1 := ExpectedString, STR2 := '] = ');
        ExpectedString := CONCAT(STR1 := ExpectedString, STR2 := BOOL_TO_STRING(Expecteds[ExpectedsIndex]));

        ActualString := 'ARRAY[';
        ActualString := CONCAT(STR1 := ActualString, STR2 := DINT_TO_STRING(ActualsIndex));
        ActualString := CONCAT(STR1 := ActualString, STR2 := '] = ');
        ActualString := CONCAT(STR1 := ActualString, STR2 := BOOL_TO_STRING(Actuals[ActualsIndex]));
    END_IF

    AssertMessageFormatter.LogAssertFailure(Expected := ExpectedString,
                                            Actual := ActualString,
                                            Message := Message,
                                            TestInstancePath := TestInstancePath);
END_IF
END_METHOD

(*
    Asserts that two BYTE arrays are equal. If they are not, an assertion error is created.
*)
METHOD PUBLIC AssertArrayEquals_BYTE
VAR_IN_OUT
    Expecteds : ARRAY[*] OF BYTE; // BYTE array with expected values
    Actuals : ARRAY[*] OF BYTE; // BYTE array with actual values
END_VAR
VAR_INPUT
    Message : Tc2_System.T_MaxString; // The identifying message for the assertion error
END_VAR
VAR
    Equals : BOOL := TRUE;
    SizeEquals : BOOL := TRUE;
    Index : DINT;
    ExpectedString : STRING;
    ActualString : STRING;
    AlreadyReported : BOOL;
    TestInstancePath : Tc2_System.T_MaxString;
    SizeOfExpecteds : DINT;
    SizeOfActuals : DINT;
    ExpectedByteString : STRING;
    ActualByteString : STRING;
    ExpectedsIndex : DINT;
    ActualsIndex : DINT;
END_VAR
IF GVL_TcUnit.IgnoreCurrentTest OR GVL_TcUnit.CurrentTestIsFinished THEN
    RETURN;
END_IF

TestInstancePath := AddTestNameToInstancePath(FindTestSuiteInstancePath());

SizeOfExpecteds := ABS(UPPER_BOUND(Expecteds, 1) - LOWER_BOUND(Expecteds, 1)) + 1;
SizeOfActuals := ABS(UPPER_BOUND(Actuals, 1) - LOWER_BOUND(Actuals, 1)) + 1;

IF SizeOfExpecteds <> SizeOfActuals THEN
    Equals := FALSE;
    SizeEquals := FALSE;
ELSE
    (* Even though we know that both arrays are equal in size, the two arrays can start at two completely different
       indexes, which needs to be taken into account for. *)
    ExpectedsIndex := LOWER_BOUND(Expecteds, 1); // The start position for the expecteds
    ActualsIndex := LOWER_BOUND(Actuals, 1); // The start position for the actuals
    FOR Index := 1 TO SizeOfExpecteds BY 1 DO
        IF Expecteds[ExpectedsIndex] <> Actuals[ActualsIndex] THEN
            Equals := FALSE;
            EXIT;
        END_IF
        ExpectedsIndex := ExpectedsIndex + 1;
        ActualsIndex := ActualsIndex + 1;
    END_FOR
END_IF

IF NOT Equals THEN
    AssertArrayResult.ReportResult(ExpectedsSize := DINT_TO_UDINT(SizeOfExpecteds),
                                   ExpectedsTypeClass := IBaseLibrary.TypeClass.TYPE_BYTE,
                                   ActualsSize := DINT_TO_UDINT(SizeOfActuals),
                                   ActualsTypeClass := IBaseLibrary.TypeClass.TYPE_BYTE,
                                   Message := Message,
                                   TestInstancePath := TestInstancePath,
                                   AlreadyReported => AlreadyReported);
END_IF

IF NOT AlreadyReported AND NOT Equals THEN
    SetTestFailed();
    
    IF NOT SizeEquals THEN
        Message := CONCAT(STR1 := Message, STR2 := ', size of arrays not matching.');
        ExpectedString := 'SIZE = ';
        ExpectedString := CONCAT(STR1 := ExpectedString, STR2 := DINT_TO_STRING(SizeOfExpecteds));
        ActualString := 'SIZE = ';
        ActualString := CONCAT(STR1 := ActualString, STR2 := DINT_TO_STRING(SizeOfActuals));
    ELSE
        ExpectedByteString := Tc2_Standard.CONCAT(STR1 := '0x',
                                                  STR2 := Tc2_Utilities.BYTE_TO_HEXSTR(in := Expecteds[ExpectedsIndex],
                                                                                       iPrecision := 2,
                                                                                       bLoCase := FALSE));
        ExpectedString := 'ARRAY[';
        ExpectedString := CONCAT(STR1 := ExpectedString, STR2 := DINT_TO_STRING(ExpectedsIndex));
        ExpectedString := CONCAT(STR1 := ExpectedString, STR2 := '] = ');
        ExpectedString := CONCAT(STR1 := ExpectedString, STR2 := ExpectedByteString);

        ActualByteString := Tc2_Standard.CONCAT(STR1 := '0x',
                                                STR2 := Tc2_Utilities.BYTE_TO_HEXSTR(in := Actuals[ActualsIndex],
                                                                                     iPrecision := 2,
                                                                                     bLoCase := FALSE));
        ActualString := 'ARRAY[';
        ActualString := CONCAT(STR1 := ActualString, STR2 := DINT_TO_STRING(ActualsIndex));
        ActualString := CONCAT(STR1 := ActualString, STR2 := '] = ');
        ActualString := CONCAT(STR1 := ActualString, STR2 := ActualByteString);
    END_IF

    AssertMessageFormatter.LogAssertFailure(Expected := ExpectedString,
                                            Actual := ActualString,
                                            Message := Message,
                                            TestInstancePath := TestInstancePath);
END_IF
END_METHOD

(*
    Asserts that two DINT arrays are equal. If they are not, an assertion error is created.
*)
METHOD PUBLIC AssertArrayEquals_DINT
VAR_IN_OUT
    Expecteds : ARRAY[*] OF DINT; // DINT array with expected values
    Actuals : ARRAY[*] OF DINT; // DINT array with actual values
END_VAR
VAR_INPUT
    Message : Tc2_System.T_MaxString; // The identifying message for the assertion error
END_VAR
VAR
    Equals : BOOL := TRUE;
    SizeEquals : BOOL := TRUE;
    Index : DINT;
    ExpectedString : STRING;
    ActualString : STRING;
    AlreadyReported : BOOL;
    TestInstancePath : Tc2_System.T_MaxString;
    SizeOfExpecteds : DINT;
    SizeOfActuals : DINT;
    ExpectedsIndex : DINT;
    ActualsIndex : DINT;
END_VAR
IF GVL_TcUnit.IgnoreCurrentTest OR GVL_TcUnit.CurrentTestIsFinished THEN
    RETURN;
END_IF

TestInstancePath := AddTestNameToInstancePath(FindTestSuiteInstancePath());

SizeOfExpecteds := ABS(UPPER_BOUND(Expecteds, 1) - LOWER_BOUND(Expecteds, 1)) + 1;
SizeOfActuals := ABS(UPPER_BOUND(Actuals, 1) - LOWER_BOUND(Actuals, 1)) + 1;

IF SizeOfExpecteds <> SizeOfActuals THEN
    Equals := FALSE;
    SizeEquals := FALSE;
ELSE
    (* Even though we know that both arrays are equal in size, the two arrays can start at two completely different
       indexes, which needs to be taken into account for. *)
    ExpectedsIndex := LOWER_BOUND(Expecteds, 1); // The start position for the expecteds
    ActualsIndex := LOWER_BOUND(Actuals, 1); // The start position for the actuals
    FOR Index := 1 TO SizeOfExpecteds BY 1 DO
        IF Expecteds[ExpectedsIndex] <> Actuals[ActualsIndex] THEN
            Equals := FALSE;
            EXIT;
        END_IF
        ExpectedsIndex := ExpectedsIndex + 1;
        ActualsIndex := ActualsIndex + 1;
    END_FOR
END_IF

IF NOT Equals THEN
    AssertArrayResult.ReportResult(ExpectedsSize := DINT_TO_UDINT(SizeOfExpecteds),
                                   ExpectedsTypeClass := IBaseLibrary.TypeClass.TYPE_DINT,
                                   ActualsSize := DINT_TO_UDINT(SizeOfActuals),
                                   ActualsTypeClass := IBaseLibrary.TypeClass.TYPE_DINT,
                                   Message := Message,
                                   TestInstancePath := TestInstancePath,
                                   AlreadyReported => AlreadyReported);
END_IF

IF NOT AlreadyReported AND NOT Equals THEN
    SetTestFailed();
    
    IF NOT SizeEquals THEN
        Message := CONCAT(STR1 := Message, STR2 := ', size of arrays not matching.');
        ExpectedString := 'SIZE = ';
        ExpectedString := CONCAT(STR1 := ExpectedString, STR2 := DINT_TO_STRING(SizeOfExpecteds));
        ActualString := 'SIZE = ';
        ActualString := CONCAT(STR1 := ActualString, STR2 := DINT_TO_STRING(SizeOfActuals));
    ELSE
        ExpectedString := 'ARRAY[';
        ExpectedString := CONCAT(STR1 := ExpectedString, STR2 := DINT_TO_STRING(ExpectedsIndex));
        ExpectedString := CONCAT(STR1 := ExpectedString, STR2 := '] = ');
        ExpectedString := CONCAT(STR1 := ExpectedString, STR2 := DINT_TO_STRING(Expecteds[ExpectedsIndex]));

        ActualString := 'ARRAY[';
        ActualString := CONCAT(STR1 := ActualString, STR2 := DINT_TO_STRING(ActualsIndex));
        ActualString := CONCAT(STR1 := ActualString, STR2 := '] = ');
        ActualString := CONCAT(STR1 := ActualString, STR2 := DINT_TO_STRING(Actuals[ActualsIndex]));
    END_IF

    AssertMessageFormatter.LogAssertFailure(Expected := ExpectedString,
                                            Actual := ActualString,
                                            Message := Message,
                                            TestInstancePath := TestInstancePath);
END_IF
END_METHOD

(*
    Asserts that two DWORD arrays are equal. If they are not, an assertion error is created.
*)
METHOD PUBLIC AssertArrayEquals_DWORD
VAR_IN_OUT
    Expecteds : ARRAY[*] OF DWORD; // DWORD array with expected values
    Actuals : ARRAY[*] OF DWORD; // DWORD array with actual values
END_VAR
VAR_INPUT
    Message : Tc2_System.T_MaxString; // The identifying message for the assertion error
END_VAR
VAR
    Equals : BOOL := TRUE;
    SizeEquals : BOOL := TRUE;
    Index : DINT;
    ExpectedString : STRING;
    ActualString : STRING;
    AlreadyReported : BOOL;
    TestInstancePath : Tc2_System.T_MaxString;
    SizeOfExpecteds : DINT;
    SizeOfActuals : DINT;
    ExpectedDWordString : STRING;
    ActualDWordString : STRING;
    ExpectedsIndex : DINT;
    ActualsIndex : DINT;
END_VAR
IF GVL_TcUnit.IgnoreCurrentTest OR GVL_TcUnit.CurrentTestIsFinished THEN
    RETURN;
END_IF

TestInstancePath := AddTestNameToInstancePath(FindTestSuiteInstancePath());

SizeOfExpecteds := ABS(UPPER_BOUND(Expecteds, 1) - LOWER_BOUND(Expecteds, 1)) + 1;
SizeOfActuals := ABS(UPPER_BOUND(Actuals, 1) - LOWER_BOUND(Actuals, 1)) + 1;

IF SizeOfExpecteds <> SizeOfActuals THEN
    Equals := FALSE;
    SizeEquals := FALSE;
ELSE
    (* Even though we know that both arrays are equal in size, the two arrays can start at two completely different
       indexes, which needs to be taken into account for. *)
    ExpectedsIndex := LOWER_BOUND(Expecteds, 1); // The start position for the expecteds
    ActualsIndex := LOWER_BOUND(Actuals, 1); // The start position for the actuals
    FOR Index := 1 TO SizeOfExpecteds BY 1 DO
        IF Expecteds[ExpectedsIndex] <> Actuals[ActualsIndex] THEN
            Equals := FALSE;
            EXIT;
        END_IF
        ExpectedsIndex := ExpectedsIndex + 1;
        ActualsIndex := ActualsIndex + 1;
    END_FOR
END_IF

IF NOT Equals THEN
    AssertArrayResult.ReportResult(ExpectedsSize := DINT_TO_UDINT(SizeOfExpecteds),
                                   ExpectedsTypeClass := IBaseLibrary.TypeClass.TYPE_DWORD,
                                   ActualsSize := DINT_TO_UDINT(SizeOfActuals),
                                   ActualsTypeClass := IBaseLibrary.TypeClass.TYPE_DWORD,
                                   Message := Message,
                                   TestInstancePath := TestInstancePath,
                                   AlreadyReported => AlreadyReported);
END_IF

IF NOT AlreadyReported AND NOT Equals THEN
    SetTestFailed();
    
    IF NOT SizeEquals THEN
        Message := CONCAT(STR1 := Message, STR2 := ', size of arrays not matching.');
        ExpectedString := 'SIZE = ';
        ExpectedString := CONCAT(STR1 := ExpectedString, STR2 := DINT_TO_STRING(SizeOfExpecteds));
        ActualString := 'SIZE = ';
        ActualString := CONCAT(STR1 := ActualString, STR2 := DINT_TO_STRING(SizeOfActuals));
    ELSE
        ExpectedDWordString := Tc2_Standard.CONCAT(STR1 := '0x',
                                                  STR2 := Tc2_Utilities.DWORD_TO_HEXSTR(in := Expecteds[ExpectedsIndex],
                                                                                        iPrecision := 8,
                                                                                        bLoCase := FALSE));
        ExpectedString := 'ARRAY[';
        ExpectedString := CONCAT(STR1 := ExpectedString, STR2 := DINT_TO_STRING(ExpectedsIndex));
        ExpectedString := CONCAT(STR1 := ExpectedString, STR2 := '] = ');
        ExpectedString := CONCAT(STR1 := ExpectedString, STR2 := ExpectedDWordString);

        ActualDWordString := Tc2_Standard.CONCAT(STR1 := '0x',
                                                STR2 := Tc2_Utilities.DWORD_TO_HEXSTR(in := Actuals[ActualsIndex],
                                                                                      iPrecision := 8,
                                                                                      bLoCase := FALSE));
        ActualString := 'ARRAY[';
        ActualString := CONCAT(STR1 := ActualString, STR2 := DINT_TO_STRING(ActualsIndex));
        ActualString := CONCAT(STR1 := ActualString, STR2 := '] = ');
        ActualString := CONCAT(STR1 := ActualString, STR2 := ActualDWordString);
    END_IF

    AssertMessageFormatter.LogAssertFailure(Expected := ExpectedString,
                                            Actual := ActualString,
                                            Message := Message,
                                            TestInstancePath := TestInstancePath);
END_IF
END_METHOD

(*
    Asserts that two INT arrays are equal. If they are not, an assertion error is created.
*)
METHOD PUBLIC AssertArrayEquals_INT
VAR_IN_OUT
    Expecteds : ARRAY[*] OF INT; // INT array with expected values
    Actuals : ARRAY[*] OF INT; // INT array with actual values
END_VAR
VAR_INPUT
    Message : Tc2_System.T_MaxString; // The identifying message for the assertion error
END_VAR
VAR
    Equals : BOOL := TRUE;
    SizeEquals : BOOL := TRUE;
    Index : DINT;
    ExpectedString : STRING;
    ActualString : STRING;
    AlreadyReported : BOOL;
    TestInstancePath : Tc2_System.T_MaxString;
    SizeOfExpecteds : DINT;
    SizeOfActuals : DINT;
    ExpectedsIndex : DINT;
    ActualsIndex : DINT;
END_VAR
IF GVL_TcUnit.IgnoreCurrentTest OR GVL_TcUnit.CurrentTestIsFinished THEN
    RETURN;
END_IF

TestInstancePath := AddTestNameToInstancePath(FindTestSuiteInstancePath());

SizeOfExpecteds := ABS(UPPER_BOUND(Expecteds, 1) - LOWER_BOUND(Expecteds, 1)) + 1;
SizeOfActuals := ABS(UPPER_BOUND(Actuals, 1) - LOWER_BOUND(Actuals, 1)) + 1;

IF SizeOfExpecteds <> SizeOfActuals THEN
    Equals := FALSE;
    SizeEquals := FALSE;
ELSE
    (* Even though we know that both arrays are equal in size, the two arrays can start at two completely different
       indexes, which needs to be taken into account for. *)
    ExpectedsIndex := LOWER_BOUND(Expecteds, 1); // The start position for the expecteds
    ActualsIndex := LOWER_BOUND(Actuals, 1); // The start position for the actuals
    FOR Index := 1 TO SizeOfExpecteds BY 1 DO
        IF Expecteds[ExpectedsIndex] <> Actuals[ActualsIndex] THEN
            Equals := FALSE;
            EXIT;
        END_IF
        ExpectedsIndex := ExpectedsIndex + 1;
        ActualsIndex := ActualsIndex + 1;
    END_FOR
END_IF

IF NOT Equals THEN
    AssertArrayResult.ReportResult(ExpectedsSize := DINT_TO_UDINT(SizeOfExpecteds),
                                   ExpectedsTypeClass := IBaseLibrary.TypeClass.TYPE_INT,
                                   ActualsSize := DINT_TO_UDINT(SizeOfActuals),
                                   ActualsTypeClass := IBaseLibrary.TypeClass.TYPE_INT,
                                   Message := Message,
                                   TestInstancePath := TestInstancePath,
                                   AlreadyReported => AlreadyReported);
END_IF

IF NOT AlreadyReported AND NOT Equals THEN
    SetTestFailed();
    
    IF NOT SizeEquals THEN
        Message := CONCAT(STR1 := Message, STR2 := ', size of arrays not matching.');
        ExpectedString := 'SIZE = ';
        ExpectedString := CONCAT(STR1 := ExpectedString, STR2 := DINT_TO_STRING(SizeOfExpecteds));
        ActualString := 'SIZE = ';
        ActualString := CONCAT(STR1 := ActualString, STR2 := DINT_TO_STRING(SizeOfActuals));
    ELSE
        ExpectedString := 'ARRAY[';
        ExpectedString := CONCAT(STR1 := ExpectedString, STR2 := DINT_TO_STRING(ExpectedsIndex));
        ExpectedString := CONCAT(STR1 := ExpectedString, STR2 := '] = ');
        ExpectedString := CONCAT(STR1 := ExpectedString, STR2 := INT_TO_STRING(Expecteds[ExpectedsIndex]));

        ActualString := 'ARRAY[';
        ActualString := CONCAT(STR1 := ActualString, STR2 := DINT_TO_STRING(ActualsIndex));
        ActualString := CONCAT(STR1 := ActualString, STR2 := '] = ');
        ActualString := CONCAT(STR1 := ActualString, STR2 := INT_TO_STRING(Actuals[ActualsIndex]));
    END_IF

    AssertMessageFormatter.LogAssertFailure(Expected := ExpectedString,
                                            Actual := ActualString,
                                            Message := Message,
                                            TestInstancePath := TestInstancePath);
END_IF
END_METHOD

(*
    Asserts that two LINT arrays are equal. If they are not, an assertion error is created.
*)
METHOD PUBLIC AssertArrayEquals_LINT
VAR_IN_OUT
    Expecteds : ARRAY[*] OF LINT; // LINT array with expected values
    Actuals : ARRAY[*] OF LINT; // LINT array with actual values
END_VAR
VAR_INPUT
    Message : Tc2_System.T_MaxString; // The identifying message for the assertion error
END_VAR
VAR
    Equals : BOOL := TRUE;
    SizeEquals : BOOL := TRUE;
    Index : DINT;
    ExpectedString : STRING;
    ActualString : STRING;
    AlreadyReported : BOOL;
    TestInstancePath : Tc2_System.T_MaxString;
    SizeOfExpecteds : DINT;
    SizeOfActuals : DINT;
    ExpectedsIndex : DINT;
    ActualsIndex : DINT;
END_VAR
IF GVL_TcUnit.IgnoreCurrentTest OR GVL_TcUnit.CurrentTestIsFinished THEN
    RETURN;
END_IF

TestInstancePath := AddTestNameToInstancePath(FindTestSuiteInstancePath());

SizeOfExpecteds := ABS(UPPER_BOUND(Expecteds, 1) - LOWER_BOUND(Expecteds, 1)) + 1;
SizeOfActuals := ABS(UPPER_BOUND(Actuals, 1) - LOWER_BOUND(Actuals, 1)) + 1;

IF SizeOfExpecteds <> SizeOfActuals THEN
    Equals := FALSE;
    SizeEquals := FALSE;
ELSE
    (* Even though we know that both arrays are equal in size, the two arrays can start at two completely different
       indexes, which needs to be taken into account for. *)
    ExpectedsIndex := LOWER_BOUND(Expecteds, 1); // The start position for the expecteds
    ActualsIndex := LOWER_BOUND(Actuals, 1); // The start position for the actuals
    FOR Index := 1 TO SizeOfExpecteds BY 1 DO
        IF Expecteds[ExpectedsIndex] <> Actuals[ActualsIndex] THEN
            Equals := FALSE;
            EXIT;
        END_IF
        ExpectedsIndex := ExpectedsIndex + 1;
        ActualsIndex := ActualsIndex + 1;
    END_FOR
END_IF

IF NOT Equals THEN
    AssertArrayResult.ReportResult(ExpectedsSize := DINT_TO_UDINT(SizeOfExpecteds),
                                   ExpectedsTypeClass := IBaseLibrary.TypeClass.TYPE_LINT,
                                   ActualsSize := DINT_TO_UDINT(SizeOfActuals),
                                   ActualsTypeClass := IBaseLibrary.TypeClass.TYPE_LINT,
                                   Message := Message,
                                   TestInstancePath := TestInstancePath,
                                   AlreadyReported => AlreadyReported);
END_IF

IF NOT AlreadyReported AND NOT Equals THEN
    SetTestFailed();
    
    IF NOT SizeEquals THEN
        Message := CONCAT(STR1 := Message, STR2 := ', size of arrays not matching.');
        ExpectedString := 'SIZE = ';
        ExpectedString := CONCAT(STR1 := ExpectedString, STR2 := DINT_TO_STRING(SizeOfExpecteds));
        ActualString := 'SIZE = ';
        ActualString := CONCAT(STR1 := ActualString, STR2 := DINT_TO_STRING(SizeOfActuals));
    ELSE
        ExpectedString := 'ARRAY[';
        ExpectedString := CONCAT(STR1 := ExpectedString, STR2 := DINT_TO_STRING(ExpectedsIndex));
        ExpectedString := CONCAT(STR1 := ExpectedString, STR2 := '] = ');
        ExpectedString := CONCAT(STR1 := ExpectedString, STR2 := LINT_TO_STRING(Expecteds[ExpectedsIndex]));

        ActualString := 'ARRAY[';
        ActualString := CONCAT(STR1 := ActualString, STR2 := DINT_TO_STRING(ActualsIndex));
        ActualString := CONCAT(STR1 := ActualString, STR2 := '] = ');
        ActualString := CONCAT(STR1 := ActualString, STR2 := LINT_TO_STRING(Actuals[ActualsIndex]));
    END_IF

    AssertMessageFormatter.LogAssertFailure(Expected := ExpectedString,
                                            Actual := ActualString,
                                            Message := Message,
                                            TestInstancePath := TestInstancePath);
END_IF
END_METHOD

METHOD PUBLIC AssertArrayEquals_LREAL
VAR_IN_OUT
    Expecteds : ARRAY[*] OF LREAL; // LREAL array with expected values
    Actuals : ARRAY[*] OF LREAL; // LREAL array with actual values
END_VAR
VAR_INPUT
    Delta : LREAL;  // The maximum delta between the value of expected and actual for which both numbers are still considered equal, proportional to the Expected value in that array cell
    Message : Tc2_System.T_MaxString; // The identifying message for the assertion error
END_VAR
VAR
    Equals : BOOL := TRUE;
    SizeEquals : BOOL := TRUE;
    Index : DINT;
    ExpectedString : STRING;
    ActualString : STRING;
    AlreadyReported : BOOL;
    TestInstancePath : Tc2_System.T_MaxString;
    SizeOfExpecteds : DINT;
    SizeOfActuals : DINT;
    ExpectedsIndex : DINT;
    ActualsIndex : DINT;
END_VAR
IF GVL_TcUnit.IgnoreCurrentTest OR GVL_TcUnit.CurrentTestIsFinished THEN
    RETURN;
END_IF

TestInstancePath := AddTestNameToInstancePath(FindTestSuiteInstancePath());

SizeOfExpecteds := ABS(UPPER_BOUND(Expecteds, 1) - LOWER_BOUND(Expecteds, 1)) + 1;
SizeOfActuals := ABS(UPPER_BOUND(Actuals, 1) - LOWER_BOUND(Actuals, 1)) + 1;

IF SizeOfExpecteds <> SizeOfActuals THEN
    Equals := FALSE;
    SizeEquals := FALSE;
ELSE
    (* Even though we know that both arrays are equal in size, the two arrays can start at two completely different
       indexes, which needs to be taken into account for. *)
    ExpectedsIndex := LOWER_BOUND(Expecteds, 1); // The start position for the expecteds
    ActualsIndex := LOWER_BOUND(Actuals, 1); // The start position for the actuals
    FOR Index := 1 TO SizeOfExpecteds BY 1 DO
        IF ABS(Expecteds[ExpectedsIndex] - Actuals[ActualsIndex]) > Delta THEN
            Equals := FALSE;
            EXIT;
        END_IF
        ExpectedsIndex := ExpectedsIndex + 1;
        ActualsIndex := ActualsIndex + 1;
    END_FOR
END_IF

IF NOT Equals THEN
    AssertArrayResult.ReportResult(ExpectedsSize := DINT_TO_UDINT(SizeOfExpecteds),
                                   ExpectedsTypeClass := IBaseLibrary.TypeClass.TYPE_LREAL,
                                   ActualsSize := DINT_TO_UDINT(SizeOfActuals),
                                   ActualsTypeClass := IBaseLibrary.TypeClass.TYPE_LREAL,
                                   Message := Message,
                                   TestInstancePath := TestInstancePath,
                                   AlreadyReported => AlreadyReported);
END_IF

IF NOT AlreadyReported AND NOT Equals THEN
    SetTestFailed();
    
    IF NOT SizeEquals THEN
        Message := CONCAT(STR1 := Message, STR2 := ', size of arrays not matching.');
        ExpectedString := 'SIZE = ';
        ExpectedString := CONCAT(STR1 := ExpectedString, STR2 := DINT_TO_STRING(SizeOfExpecteds));
        ActualString := 'SIZE = ';
        ActualString := CONCAT(STR1 := ActualString, STR2 := DINT_TO_STRING(SizeOfActuals));
    ELSE
        ExpectedString := 'ARRAY[';
        ExpectedString := CONCAT(STR1 := ExpectedString, STR2 := DINT_TO_STRING(ExpectedsIndex));
        ExpectedString := CONCAT(STR1 := ExpectedString, STR2 := '] = ');
        ExpectedString := CONCAT(STR1 := ExpectedString, STR2 := LREAL_TO_STRING(Expecteds[ExpectedsIndex]));

        ActualString := 'ARRAY[';
        ActualString := CONCAT(STR1 := ActualString, STR2 := DINT_TO_STRING(ActualsIndex));
        ActualString := CONCAT(STR1 := ActualString, STR2 := '] = ');
        ActualString := CONCAT(STR1 := ActualString, STR2 := LREAL_TO_STRING(Actuals[ActualsIndex]));
    END_IF

    AssertMessageFormatter.LogAssertFailure(Expected := ExpectedString,
                                            Actual := ActualString,
                                            Message := Message,
                                            TestInstancePath := TestInstancePath);
END_IF
END_METHOD

(*
    Asserts that two LWORD arrays are equal. If they are not, an assertion error is created.
*)
METHOD PUBLIC AssertArrayEquals_LWORD
VAR_IN_OUT
    Expecteds : ARRAY[*] OF LWORD; // LWORD array with expected values
    Actuals : ARRAY[*] OF LWORD; // LWORD array with actual values
END_VAR
VAR_INPUT
    Message : Tc2_System.T_MaxString; // The identifying message for the assertion error
END_VAR
VAR
    Equals : BOOL := TRUE;
    SizeEquals : BOOL := TRUE;
    Index : DINT;
    ExpectedString : STRING;
    ActualString : STRING;
    AlreadyReported : BOOL;
    TestInstancePath : Tc2_System.T_MaxString;
    SizeOfExpecteds : DINT;
    SizeOfActuals : DINT;
    ExpectedDWordString : STRING;
    ActualDWordString : STRING;
    ExpectedsIndex : DINT;
    ActualsIndex : DINT;
END_VAR
IF GVL_TcUnit.IgnoreCurrentTest OR GVL_TcUnit.CurrentTestIsFinished THEN
    RETURN;
END_IF

TestInstancePath := AddTestNameToInstancePath(FindTestSuiteInstancePath());

SizeOfExpecteds := ABS(UPPER_BOUND(Expecteds, 1) - LOWER_BOUND(Expecteds, 1)) + 1;
SizeOfActuals := ABS(UPPER_BOUND(Actuals, 1) - LOWER_BOUND(Actuals, 1)) + 1;

IF SizeOfExpecteds <> SizeOfActuals THEN
    Equals := FALSE;
    SizeEquals := FALSE;
ELSE
    (* Even though we know that both arrays are equal in size, the two arrays can start at two completely different
       indexes, which needs to be taken into account for. *)
    ExpectedsIndex := LOWER_BOUND(Expecteds, 1); // The start position for the expecteds
    ActualsIndex := LOWER_BOUND(Actuals, 1); // The start position for the actuals
    FOR Index := 1 TO SizeOfExpecteds BY 1 DO
        IF Expecteds[ExpectedsIndex] <> Actuals[ActualsIndex] THEN
            Equals := FALSE;
            EXIT;
        END_IF
        ExpectedsIndex := ExpectedsIndex + 1;
        ActualsIndex := ActualsIndex + 1;
    END_FOR
END_IF

IF NOT Equals THEN
    AssertArrayResult.ReportResult(ExpectedsSize := DINT_TO_UDINT(SizeOfExpecteds),
                                   ExpectedsTypeClass := IBaseLibrary.TypeClass.TYPE_LWORD,
                                   ActualsSize := DINT_TO_UDINT(SizeOfActuals),
                                   ActualsTypeClass := IBaseLibrary.TypeClass.TYPE_LWORD,
                                   Message := Message,
                                   TestInstancePath := TestInstancePath,
                                   AlreadyReported => AlreadyReported);
END_IF

IF NOT AlreadyReported AND NOT Equals THEN
    SetTestFailed();
    
    IF NOT SizeEquals THEN
        Message := CONCAT(STR1 := Message, STR2 := ', size of arrays not matching.');
        ExpectedString := 'SIZE = ';
        ExpectedString := CONCAT(STR1 := ExpectedString, STR2 := DINT_TO_STRING(SizeOfExpecteds));
        ActualString := 'SIZE = ';
        ActualString := CONCAT(STR1 := ActualString, STR2 := DINT_TO_STRING(SizeOfActuals));
    ELSE
        ExpectedDWordString := Tc2_Standard.CONCAT(STR1 := '0x',
                                                  STR2 := Tc2_Utilities.LWORD_TO_HEXSTR(in := Expecteds[ExpectedsIndex],
                                                                                        iPrecision := 16,
                                                                                        bLoCase := FALSE));
        ExpectedString := 'ARRAY[';
        ExpectedString := CONCAT(STR1 := ExpectedString, STR2 := DINT_TO_STRING(ExpectedsIndex));
        ExpectedString := CONCAT(STR1 := ExpectedString, STR2 := '] = ');
        ExpectedString := CONCAT(STR1 := ExpectedString, STR2 := ExpectedDWordString);

        ActualDWordString := Tc2_Standard.CONCAT(STR1 := '0x',
                                                STR2 := Tc2_Utilities.LWORD_TO_HEXSTR(in := Actuals[ActualsIndex],
                                                                                      iPrecision := 16,
                                                                                      bLoCase := FALSE));
        ActualString := 'ARRAY[';
        ActualString := CONCAT(STR1 := ActualString, STR2 := DINT_TO_STRING(ActualsIndex));
        ActualString := CONCAT(STR1 := ActualString, STR2 := '] = ');
        ActualString := CONCAT(STR1 := ActualString, STR2 := ActualDWordString);
    END_IF

    AssertMessageFormatter.LogAssertFailure(Expected := ExpectedString,
                                            Actual := ActualString,
                                            Message := Message,
                                            TestInstancePath := TestInstancePath);
END_IF
END_METHOD

METHOD PUBLIC AssertArrayEquals_REAL
VAR_IN_OUT
    Expecteds : ARRAY[*] OF REAL; // REAL array with expected values
    Actuals : ARRAY[*] OF REAL; // REAL array with actual values
END_VAR
VAR_INPUT
    Delta : REAL;  // The maximum delta between the value of expected and actual for which both numbers are still considered equal, proportional to the Expected value in that array cell
    Message : Tc2_System.T_MaxString; // The identifying message for the assertion error
END_VAR
VAR
    Equals : BOOL := TRUE;
    SizeEquals : BOOL := TRUE;
    Index : DINT;
    ExpectedString : STRING;
    ActualString : STRING;
    AlreadyReported : BOOL;
    TestInstancePath : Tc2_System.T_MaxString;
    SizeOfExpecteds : DINT;
    SizeOfActuals : DINT;
    ExpectedsIndex : DINT;
    ActualsIndex : DINT;
END_VAR
IF GVL_TcUnit.IgnoreCurrentTest OR GVL_TcUnit.CurrentTestIsFinished THEN
    RETURN;
END_IF

TestInstancePath := AddTestNameToInstancePath(FindTestSuiteInstancePath());

SizeOfExpecteds := ABS(UPPER_BOUND(Expecteds, 1) - LOWER_BOUND(Expecteds, 1)) + 1;
SizeOfActuals := ABS(UPPER_BOUND(Actuals, 1) - LOWER_BOUND(Actuals, 1)) + 1;

IF SizeOfExpecteds <> SizeOfActuals THEN
    Equals := FALSE;
    SizeEquals := FALSE;
ELSE
    (* Even though we know that both arrays are equal in size, the two arrays can start at two completely different
       indexes, which needs to be taken into account for. *)
    ExpectedsIndex := LOWER_BOUND(Expecteds, 1); // The start position for the expecteds
    ActualsIndex := LOWER_BOUND(Actuals, 1); // The start position for the actuals
    FOR Index := 1 TO SizeOfExpecteds BY 1 DO
        IF ABS(Expecteds[ExpectedsIndex] - Actuals[ActualsIndex]) > Delta THEN
            Equals := FALSE;
            EXIT;
        END_IF
        ExpectedsIndex := ExpectedsIndex + 1;
        ActualsIndex := ActualsIndex + 1;
    END_FOR
END_IF

IF NOT Equals THEN
    AssertArrayResult.ReportResult(ExpectedsSize := DINT_TO_UDINT(SizeOfExpecteds),
                                   ExpectedsTypeClass := IBaseLibrary.TypeClass.TYPE_REAL,
                                   ActualsSize := DINT_TO_UDINT(SizeOfActuals),
                                   ActualsTypeClass := IBaseLibrary.TypeClass.TYPE_REAL,
                                   Message := Message,
                                   TestInstancePath := TestInstancePath,
                                   AlreadyReported => AlreadyReported);
END_IF

IF NOT AlreadyReported AND NOT Equals THEN
    SetTestFailed();
    
    IF NOT SizeEquals THEN
        Message := CONCAT(STR1 := Message, STR2 := ', size of arrays not matching.');
        ExpectedString := 'SIZE = ';
        ExpectedString := CONCAT(STR1 := ExpectedString, STR2 := DINT_TO_STRING(SizeOfExpecteds));
        ActualString := 'SIZE = ';
        ActualString := CONCAT(STR1 := ActualString, STR2 := DINT_TO_STRING(SizeOfActuals));
    ELSE
        ExpectedString := 'ARRAY[';
        ExpectedString := CONCAT(STR1 := ExpectedString, STR2 := DINT_TO_STRING(ExpectedsIndex));
        ExpectedString := CONCAT(STR1 := ExpectedString, STR2 := '] = ');
        ExpectedString := CONCAT(STR1 := ExpectedString, STR2 := REAL_TO_STRING(Expecteds[ExpectedsIndex]));

        ActualString := 'ARRAY[';
        ActualString := CONCAT(STR1 := ActualString, STR2 := DINT_TO_STRING(ActualsIndex));
        ActualString := CONCAT(STR1 := ActualString, STR2 := '] = ');
        ActualString := CONCAT(STR1 := ActualString, STR2 := REAL_TO_STRING(Actuals[ActualsIndex]));
    END_IF

    AssertMessageFormatter.LogAssertFailure(Expected := ExpectedString,
                                            Actual := ActualString,
                                            Message := Message,
                                            TestInstancePath := TestInstancePath);
END_IF
END_METHOD

(*
    Asserts that two SINT arrays are equal. If they are not, an assertion error is created.
*)
METHOD PUBLIC AssertArrayEquals_SINT
VAR_IN_OUT
    Expecteds : ARRAY[*] OF SINT; // SINT array with expected values
    Actuals : ARRAY[*] OF SINT; // SINT array with actual values
END_VAR
VAR_INPUT
    Message : Tc2_System.T_MaxString; // The identifying message for the assertion error
END_VAR
VAR
    Equals : BOOL := TRUE;
    SizeEquals : BOOL := TRUE;
    Index : DINT;
    ExpectedString : STRING;
    ActualString : STRING;
    AlreadyReported : BOOL;
    TestInstancePath : Tc2_System.T_MaxString;
    SizeOfExpecteds : DINT;
    SizeOfActuals : DINT;
    ExpectedsIndex : DINT;
    ActualsIndex : DINT;
END_VAR
IF GVL_TcUnit.IgnoreCurrentTest OR GVL_TcUnit.CurrentTestIsFinished THEN
    RETURN;
END_IF

TestInstancePath := AddTestNameToInstancePath(FindTestSuiteInstancePath());

SizeOfExpecteds := ABS(UPPER_BOUND(Expecteds, 1) - LOWER_BOUND(Expecteds, 1)) + 1;
SizeOfActuals := ABS(UPPER_BOUND(Actuals, 1) - LOWER_BOUND(Actuals, 1)) + 1;

IF SizeOfExpecteds <> SizeOfActuals THEN
    Equals := FALSE;
    SizeEquals := FALSE;
ELSE
    (* Even though we know that both arrays are equal in size, the two arrays can start at two completely different
       indexes, which needs to be taken into account for. *)
    ExpectedsIndex := LOWER_BOUND(Expecteds, 1); // The start position for the expecteds
    ActualsIndex := LOWER_BOUND(Actuals, 1); // The start position for the actuals
    FOR Index := 1 TO SizeOfExpecteds BY 1 DO
        IF Expecteds[ExpectedsIndex] <> Actuals[ActualsIndex] THEN
            Equals := FALSE;
            EXIT;
        END_IF
        ExpectedsIndex := ExpectedsIndex + 1;
        ActualsIndex := ActualsIndex + 1;
    END_FOR
END_IF

IF NOT Equals THEN
    AssertArrayResult.ReportResult(ExpectedsSize := DINT_TO_UDINT(SizeOfExpecteds),
                                   ExpectedsTypeClass := IBaseLibrary.TypeClass.TYPE_SINT,
                                   ActualsSize := DINT_TO_UDINT(SizeOfActuals),
                                   ActualsTypeClass := IBaseLibrary.TypeClass.TYPE_SINT,
                                   Message := Message,
                                   TestInstancePath := TestInstancePath,
                                   AlreadyReported => AlreadyReported);
END_IF

IF NOT AlreadyReported AND NOT Equals THEN
    SetTestFailed();
    
    IF NOT SizeEquals THEN
        Message := CONCAT(STR1 := Message, STR2 := ', size of arrays not matching.');
        ExpectedString := 'SIZE = ';
        ExpectedString := CONCAT(STR1 := ExpectedString, STR2 := DINT_TO_STRING(SizeOfExpecteds));
        ActualString := 'SIZE = ';
        ActualString := CONCAT(STR1 := ActualString, STR2 := DINT_TO_STRING(SizeOfActuals));
    ELSE
        ExpectedString := 'ARRAY[';
        ExpectedString := CONCAT(STR1 := ExpectedString, STR2 := DINT_TO_STRING(ExpectedsIndex));
        ExpectedString := CONCAT(STR1 := ExpectedString, STR2 := '] = ');
        ExpectedString := CONCAT(STR1 := ExpectedString, STR2 := SINT_TO_STRING(Expecteds[ExpectedsIndex]));

        ActualString := 'ARRAY[';
        ActualString := CONCAT(STR1 := ActualString, STR2 := DINT_TO_STRING(ActualsIndex));
        ActualString := CONCAT(STR1 := ActualString, STR2 := '] = ');
        ActualString := CONCAT(STR1 := ActualString, STR2 := SINT_TO_STRING(Actuals[ActualsIndex]));
    END_IF

    AssertMessageFormatter.LogAssertFailure(Expected := ExpectedString,
                                            Actual := ActualString,
                                            Message := Message,
                                            TestInstancePath := TestInstancePath);
END_IF
END_METHOD

(*
    Asserts that two UDINT arrays are equal. If they are not, an assertion error is created.
*)
METHOD PUBLIC AssertArrayEquals_UDINT
VAR_IN_OUT
    Expecteds : ARRAY[*] OF UDINT; // UDINT array with expected values
    Actuals : ARRAY[*] OF UDINT; // UDINT array with actual values
END_VAR
VAR_INPUT
    Message : Tc2_System.T_MaxString; // The identifying message for the assertion error
END_VAR
VAR
    Equals : BOOL := TRUE;
    SizeEquals : BOOL := TRUE;
    Index : DINT;
    ExpectedString : STRING;
    ActualString : STRING;
    AlreadyReported : BOOL;
    TestInstancePath : Tc2_System.T_MaxString;
    SizeOfExpecteds : DINT;
    SizeOfActuals : DINT;
    ExpectedsIndex : DINT;
    ActualsIndex : DINT;
END_VAR
IF GVL_TcUnit.IgnoreCurrentTest OR GVL_TcUnit.CurrentTestIsFinished THEN
    RETURN;
END_IF

TestInstancePath := AddTestNameToInstancePath(FindTestSuiteInstancePath());

SizeOfExpecteds := ABS(UPPER_BOUND(Expecteds, 1) - LOWER_BOUND(Expecteds, 1)) + 1;
SizeOfActuals := ABS(UPPER_BOUND(Actuals, 1) - LOWER_BOUND(Actuals, 1)) + 1;

IF SizeOfExpecteds <> SizeOfActuals THEN
    Equals := FALSE;
    SizeEquals := FALSE;
ELSE
    (* Even though we know that both arrays are equal in size, the two arrays can start at two completely different
       indexes, which needs to be taken into account for. *)
    ExpectedsIndex := LOWER_BOUND(Expecteds, 1); // The start position for the expecteds
    ActualsIndex := LOWER_BOUND(Actuals, 1); // The start position for the actuals
    FOR Index := 1 TO SizeOfExpecteds BY 1 DO
        IF Expecteds[ExpectedsIndex] <> Actuals[ActualsIndex] THEN
            Equals := FALSE;
            EXIT;
        END_IF
        ExpectedsIndex := ExpectedsIndex + 1;
        ActualsIndex := ActualsIndex + 1;
    END_FOR
END_IF

IF NOT Equals THEN
    AssertArrayResult.ReportResult(ExpectedsSize := DINT_TO_UDINT(SizeOfExpecteds),
                                   ExpectedsTypeClass := IBaseLibrary.TypeClass.TYPE_UDINT,
                                   ActualsSize := DINT_TO_UDINT(SizeOfActuals),
                                   ActualsTypeClass := IBaseLibrary.TypeClass.TYPE_UDINT,
                                   Message := Message,
                                   TestInstancePath := TestInstancePath,
                                   AlreadyReported => AlreadyReported);
END_IF

IF NOT AlreadyReported AND NOT Equals THEN
    SetTestFailed();
    
    IF NOT SizeEquals THEN
        Message := CONCAT(STR1 := Message, STR2 := ', size of arrays not matching.');
        ExpectedString := 'SIZE = ';
        ExpectedString := CONCAT(STR1 := ExpectedString, STR2 := DINT_TO_STRING(SizeOfExpecteds));
        ActualString := 'SIZE = ';
        ActualString := CONCAT(STR1 := ActualString, STR2 := DINT_TO_STRING(SizeOfActuals));
    ELSE
        ExpectedString := 'ARRAY[';
        ExpectedString := CONCAT(STR1 := ExpectedString, STR2 := DINT_TO_STRING(ExpectedsIndex));
        ExpectedString := CONCAT(STR1 := ExpectedString, STR2 := '] = ');
        ExpectedString := CONCAT(STR1 := ExpectedString, STR2 := UDINT_TO_STRING(Expecteds[ExpectedsIndex]));

        ActualString := 'ARRAY[';
        ActualString := CONCAT(STR1 := ActualString, STR2 := DINT_TO_STRING(ActualsIndex));
        ActualString := CONCAT(STR1 := ActualString, STR2 := '] = ');
        ActualString := CONCAT(STR1 := ActualString, STR2 := UDINT_TO_STRING(Actuals[ActualsIndex]));
    END_IF

    AssertMessageFormatter.LogAssertFailure(Expected := ExpectedString,
                                            Actual := ActualString,
                                            Message := Message,
                                            TestInstancePath := TestInstancePath);
END_IF
END_METHOD

(*
    Asserts that two UINT arrays are equal. If they are not, an assertion error is created.
*)
METHOD PUBLIC AssertArrayEquals_UINT
VAR_IN_OUT
    Expecteds : ARRAY[*] OF UINT; // UINT array with expected values
    Actuals : ARRAY[*] OF UINT; // UINT array with actual values
END_VAR
VAR_INPUT
    Message : Tc2_System.T_MaxString; // The identifying message for the assertion error
END_VAR
VAR
    Equals : BOOL := TRUE;
    SizeEquals : BOOL := TRUE;
    Index : DINT;
    ExpectedString : STRING;
    ActualString : STRING;
    AlreadyReported : BOOL;
    TestInstancePath : Tc2_System.T_MaxString;
    SizeOfExpecteds : DINT;
    SizeOfActuals : DINT;
    ExpectedsIndex : DINT;
    ActualsIndex : DINT;
END_VAR
IF GVL_TcUnit.IgnoreCurrentTest OR GVL_TcUnit.CurrentTestIsFinished THEN
    RETURN;
END_IF

TestInstancePath := AddTestNameToInstancePath(FindTestSuiteInstancePath());

SizeOfExpecteds := ABS(UPPER_BOUND(Expecteds, 1) - LOWER_BOUND(Expecteds, 1)) + 1;
SizeOfActuals := ABS(UPPER_BOUND(Actuals, 1) - LOWER_BOUND(Actuals, 1)) + 1;

IF SizeOfExpecteds <> SizeOfActuals THEN
    Equals := FALSE;
    SizeEquals := FALSE;
ELSE
    (* Even though we know that both arrays are equal in size, the two arrays can start at two completely different
       indexes, which needs to be taken into account for. *)
    ExpectedsIndex := LOWER_BOUND(Expecteds, 1); // The start position for the expecteds
    ActualsIndex := LOWER_BOUND(Actuals, 1); // The start position for the actuals
    FOR Index := 1 TO SizeOfExpecteds BY 1 DO
        IF Expecteds[ExpectedsIndex] <> Actuals[ActualsIndex] THEN
            Equals := FALSE;
            EXIT;
        END_IF
        ExpectedsIndex := ExpectedsIndex + 1;
        ActualsIndex := ActualsIndex + 1;
    END_FOR
END_IF

IF NOT Equals THEN
    AssertArrayResult.ReportResult(ExpectedsSize := DINT_TO_UDINT(SizeOfExpecteds),
                                   ExpectedsTypeClass := IBaseLibrary.TypeClass.TYPE_UINT,
                                   ActualsSize := DINT_TO_UDINT(SizeOfActuals),
                                   ActualsTypeClass := IBaseLibrary.TypeClass.TYPE_UINT,
                                   Message := Message,
                                   TestInstancePath := TestInstancePath,
                                   AlreadyReported => AlreadyReported);
END_IF

IF NOT AlreadyReported AND NOT Equals THEN
    SetTestFailed();
    
    IF NOT SizeEquals THEN
        Message := CONCAT(STR1 := Message, STR2 := ', size of arrays not matching.');
        ExpectedString := 'SIZE = ';
        ExpectedString := CONCAT(STR1 := ExpectedString, STR2 := DINT_TO_STRING(SizeOfExpecteds));
        ActualString := 'SIZE = ';
        ActualString := CONCAT(STR1 := ActualString, STR2 := DINT_TO_STRING(SizeOfActuals));
    ELSE
        ExpectedString := 'ARRAY[';
        ExpectedString := CONCAT(STR1 := ExpectedString, STR2 := DINT_TO_STRING(ExpectedsIndex));
        ExpectedString := CONCAT(STR1 := ExpectedString, STR2 := '] = ');
        ExpectedString := CONCAT(STR1 := ExpectedString, STR2 := UINT_TO_STRING(Expecteds[ExpectedsIndex]));

        ActualString := 'ARRAY[';
        ActualString := CONCAT(STR1 := ActualString, STR2 := DINT_TO_STRING(ActualsIndex));
        ActualString := CONCAT(STR1 := ActualString, STR2 := '] = ');
        ActualString := CONCAT(STR1 := ActualString, STR2 := UINT_TO_STRING(Actuals[ActualsIndex]));
    END_IF

    AssertMessageFormatter.LogAssertFailure(Expected := ExpectedString,
                                            Actual := ActualString,
                                            Message := Message,
                                            TestInstancePath := TestInstancePath);
END_IF
END_METHOD

(*
    Asserts that two ULINT arrays are equal. If they are not, an assertion error is created.
*)
METHOD PUBLIC AssertArrayEquals_ULINT
VAR_IN_OUT
    Expecteds : ARRAY[*] OF ULINT; // ULINT array with expected values
    Actuals : ARRAY[*] OF ULINT; // ULINT array with actual values
END_VAR
VAR_INPUT
    Message : Tc2_System.T_MaxString; // The identifying message for the assertion error
END_VAR
VAR
    Equals : BOOL := TRUE;
    SizeEquals : BOOL := TRUE;
    Index : DINT;
    ExpectedString : STRING;
    ActualString : STRING;
    AlreadyReported : BOOL;
    TestInstancePath : Tc2_System.T_MaxString;
    SizeOfExpecteds : DINT;
    SizeOfActuals : DINT;
    ExpectedsIndex : DINT;
    ActualsIndex : DINT;
END_VAR
IF GVL_TcUnit.IgnoreCurrentTest OR GVL_TcUnit.CurrentTestIsFinished THEN
    RETURN;
END_IF

TestInstancePath := AddTestNameToInstancePath(FindTestSuiteInstancePath());

SizeOfExpecteds := ABS(UPPER_BOUND(Expecteds, 1) - LOWER_BOUND(Expecteds, 1)) + 1;
SizeOfActuals := ABS(UPPER_BOUND(Actuals, 1) - LOWER_BOUND(Actuals, 1)) + 1;

IF SizeOfExpecteds <> SizeOfActuals THEN
    Equals := FALSE;
    SizeEquals := FALSE;
ELSE
    (* Even though we know that both arrays are equal in size, the two arrays can start at two completely different
       indexes, which needs to be taken into account for. *)
    ExpectedsIndex := LOWER_BOUND(Expecteds, 1); // The start position for the expecteds
    ActualsIndex := LOWER_BOUND(Actuals, 1); // The start position for the actuals
    FOR Index := 1 TO SizeOfExpecteds BY 1 DO
        IF Expecteds[ExpectedsIndex] <> Actuals[ActualsIndex] THEN
            Equals := FALSE;
            EXIT;
        END_IF
        ExpectedsIndex := ExpectedsIndex + 1;
        ActualsIndex := ActualsIndex + 1;
    END_FOR
END_IF

IF NOT Equals THEN
    AssertArrayResult.ReportResult(ExpectedsSize := DINT_TO_UDINT(SizeOfExpecteds),
                                   ExpectedsTypeClass := IBaseLibrary.TypeClass.TYPE_ULINT,
                                   ActualsSize := DINT_TO_UDINT(SizeOfActuals),
                                   ActualsTypeClass := IBaseLibrary.TypeClass.TYPE_ULINT,
                                   Message := Message,
                                   TestInstancePath := TestInstancePath,
                                   AlreadyReported => AlreadyReported);
END_IF

IF NOT AlreadyReported AND NOT Equals THEN
    SetTestFailed();
    
    IF NOT SizeEquals THEN
        Message := CONCAT(STR1 := Message, STR2 := ', size of arrays not matching.');
        ExpectedString := 'SIZE = ';
        ExpectedString := CONCAT(STR1 := ExpectedString, STR2 := DINT_TO_STRING(SizeOfExpecteds));
        ActualString := 'SIZE = ';
        ActualString := CONCAT(STR1 := ActualString, STR2 := DINT_TO_STRING(SizeOfActuals));
    ELSE
        ExpectedString := 'ARRAY[';
        ExpectedString := CONCAT(STR1 := ExpectedString, STR2 := DINT_TO_STRING(ExpectedsIndex));
        ExpectedString := CONCAT(STR1 := ExpectedString, STR2 := '] = ');
        ExpectedString := CONCAT(STR1 := ExpectedString, STR2 := ULINT_TO_STRING(Expecteds[ExpectedsIndex]));

        ActualString := 'ARRAY[';
        ActualString := CONCAT(STR1 := ActualString, STR2 := DINT_TO_STRING(ActualsIndex));
        ActualString := CONCAT(STR1 := ActualString, STR2 := '] = ');
        ActualString := CONCAT(STR1 := ActualString, STR2 := ULINT_TO_STRING(Actuals[ActualsIndex]));
    END_IF

